(* Logix 5000 project; controller PBS_Perfusion vendor 1 type 14 code 217 rev 32.14; software revision 32.03; part 24 of 27 *)
(* tags used below, declared in another part *)
   Inp_Ready : BOOL;   // 1=Drive is ready to run
   Inp_CommandDir : BOOL;   // 1=Drive is commanded Forward, 0=Drive is commanded Reverse
   Inp_ActualDir : BOOL;   // 1=Drive is running Forward, 0=Drive is running Reverse
   Inp_FwdPermOK : BOOL;   // 1=Permissives OK, drive can start Forward
   Inp_FwdNBPermOK : BOOL;   // 1=Non-Bypassable Permissives OK, drive can start Forward
   Inp_RevPermOK : BOOL;   // 1=Permissives OK, drive can start Reverse
   Inp_RevNBPermOK : BOOL;   // 1=Non-Bypassable Permissives OK, motor can start Reverse
   Inp_IntlkOK : BOOL;   // 1=Interlocks OK, drive can start/run
   Inp_NBIntlkOK : BOOL;   // 1=Non-Bypassable Interlocks OK, drive can start/run
   Inp_OvrdCmd : DINT;   // Override Command: 0=None, 1=Stop, 2=Start Fwd 3=Start Rev
   Cfg_HasReverse : BOOL;   // 1=Drive can be run reverse, 0=Forward only
   Cfg_HasIntlkObj : BOOL;   // 1=Tells HMI a P_Intlk is connected to Inp_Intlk
   Cfg_SetTrack : BOOL;   // 1=Settings track for unselected sources, 0=no tracking
   Cfg_ShedOnFailToStart : BOOL;   // 1=Stop Motor and Alarm on Fail to Start; 0=Alarm only on Fail to Start
   Cfg_ShedOnIOFault : BOOL;   // 1=Stop Motor and Alarm on I/O Fault; 0=Alarm only on I/O Fault
   Cfg_DecPlcs : DINT;   // Number of decimal places for speed ref/fdbk display (0..6)
   Cfg_InpDLDecPlcs : DINT;   // Number of decimal places for Input Datalink display (0..6)
   Cfg_OutDLDecPlcs : DINT;   // Number of decimal places for Output Datalink display (0..6)
   Cfg_FailToStartAckReqd : ALIAS FOR FailToStart.Cfg_AckReqd;   // 1=Acknowledge required for Fail to Start Alarm
   Cfg_FailToStopAckReqd : ALIAS FOR FailToStop.Cfg_AckReqd;   // 1=Acknowledge required for Fail to Stop Alarm
   Cfg_IntlkTripAckReqd : ALIAS FOR IntlkTrip.Cfg_AckReqd;   // 1=Acknowledge required for Interlock Trip Alarm
   Cfg_DriveFaultAckReqd : ALIAS FOR DriveFault.Cfg_AckReqd;   // 1=Acknowledge required for Drive Fault Alarm
   Cfg_IOFaultAckReqd : ALIAS FOR IOFault.Cfg_AckReqd;   // 1=Acknowledge required for I/O Fault Alarm
   Cfg_FailToStartSeverity : ALIAS FOR FailToStart.Cfg_Severity;   // Fail To Start Alarm Severity: 1..250=Low, 251..500=Medium, 501..750=High, 751..1000=Urgent
   Cfg_FailToStopSeverity : ALIAS FOR FailToStop.Cfg_Severity;   // Fail To Stop Alarm Severity: 1..250=Low, 251..500=Medium, 501..750=High, 751..1000=Urgent
   Cfg_IntlkTripSeverity : ALIAS FOR IntlkTrip.Cfg_Severity;   // Interlock Trip Alarm Severity: 1..250=Low, 251..500=Medium, 501..750=High, 751..1000=Urgent
   Cfg_DriveFaultSeverity : ALIAS FOR DriveFault.Cfg_Severity;   // Drive Fault Alarm Severity: 1..250=Low, 251..500=Medium, 501..750=High, 751..1000=Urgent
   Cfg_IOFaultSeverity : ALIAS FOR IOFault.Cfg_Severity;   // I/O Fault Alarm Severity: 1..250=Low, 251..500=Medium, 501..750=High, 751..1000=Urgent
   Cfg_MaxSpdRef : REAL;   // Maximum Speed Reference in EU (for limiting)
   Cfg_SpeedRefRawMax : REAL;   // Speed Reference Maximum in Drive (raw) Units (for scaling)
   Cfg_SpeedRefEUMax : REAL;   // Speed Reference Maximum in Engineering Units (for scaling)
   Cfg_SpeedFdbkRawMax : REAL;   // Speed Feedback Maximum in Drive (raw) Units (for scaling)
   Cfg_SpeedFdbkEUMax : REAL;   // Speed Feedback Maximum in Engineering Units (for scaling)
   Cfg_InpDatalinkRawMax : REAL;   // Input Datalink Maximum in Drive (raw) Units (for scaling)
   Cfg_InpDatalinkEUMax : REAL;   // Input Datalink Maximum in Engineering Units (for scaling)
   Cfg_OutDatalinkMax : REAL;   // Maximum Output Datalink in EU (for limiting)
   Cfg_OutDatalinkRawMax : REAL;   // Output Datalink Maximum in Drive (raw) Units (for scaling)
   Cfg_OutDatalinkEUMax : REAL;   // Output Datalink Maximum in Engineering Units (for scaling)
   Cfg_SimRampT : REAL;   // Time to ramp speed fdbk when in Simulation (sec)
   Cfg_FailToStartT : REAL;   // Time after Start to get Run Feedback before Fault (sec)
   Cfg_FailToStopT : REAL;   // Time after Stop to drop Run Feedback before Fault (sec)
   Cfg_ResetPulseT : REAL;   // Time to pulse Out_Reset to clear drive fault
   Cfg_OperKeep : SINT;   // Oper keeps control in Prog / Ext: .0=Reference, .1=Start/Stop/Fwd/ Rev, .3=OutDatalink
   Cfg_ProgKeep : SINT;   // Prog keeps control in Oper / Ext: .0=Reference, .1=Start/Stop/Fwd/ Rev, .3=OutDatalink
   Cfg_ExtKeep : SINT;   // Ext keeps control in Prog / Oper: .0=Reference, .1=Start/Stop/Fwd/ Rev, .3=OutDatalink
   PSet_SpeedRef : REAL;   // Program Setting of Speed Reference (EU)
   PSet_Owner : DINT;   // Program Owner Request ID (non-zero) or Release (zero)
   XSet_SpeedRef : REAL;   // External Setting of Speed Reference (EU)
   PCmd_StartFwd : BOOL;   // Program Command to Start Drive Forward
   PCmd_StartRev : BOOL;   // Program Command to Start Drive Reverse
   PCmd_Stop : BOOL;   // Program Command to Stop Drive
   PCmd_Reset : BOOL;   // Program Command to Reset drive fault and all Alarms requiring Reset
   XCmd_StartFwd : BOOL;   // External Command to Start Drive Forward
   XCmd_StartRev : BOOL;   // External Command to Start Drive Reverse
   XCmd_Stop : BOOL;   // External Command to Stop Drive
   XCmd_JogFwd : BOOL;   // External Command to Jog Drive Forward
   XCmd_JogRev : BOOL;   // External Command to Jog Drive Reverse
   XCmd_Reset : BOOL;   // Ext Cmd to clear shed latches and cleared alarms
   Out_SpeedRef : REAL;   // Drive Speed Reference in Drive Units (typ. 0-32767 = 0 to max freq.)
   Out_Datalink : REAL;   // Auxiliary Signal (datalink) Output in Drive (raw) Units
   Out_Run : BOOL;   // 1=Start/Run Drive, 0=Stop Drive (for held starter type)
   Out_Stop : BOOL;   // 1=Stop Drive, 0=drive left in current state
   Out_Start : BOOL;   // 1=Start Drive, 0=drive left in current state
   Out_Jog : BOOL;   // 1=Jog drive at Jog Speed, -->0=stop jogging
   Out_ClearFault : BOOL;   // 1=Attempt to clear Drive Fault
   Out_Fwd : BOOL;   // 1=Set drive direction to Forward
   Out_Rev : BOOL;   // 1=Set drive direction to Reverse
   Out_Horn : BOOL;   // 1=Sound audible prior to commanded motor start
   Val_SpeedRef : REAL;   // Speed Reference (target) to drive
   Val_SpeedRefEUMax : REAL;   // Maximum of Speed Reference = MAX (Cfg_SpeedFdbkEUMin, Cfg_SpeedFdbkEUMax)
   Val_SpeedFdbkEUMax : REAL;   // Maximum of Speed Feedback = MAX (Cfg_SpeedFdbkEUMin, Cfg_SpeedFdbkEUMax)
   SrcQ_IO : DINT;   // Source and Quality of primary I/O (enumeration)
   SrcQ : DINT;   // Source and Quality of primary Val/Sts (enumeration)
   Val_Cmd : DINT;   // Device Command 0=None, 1=Stop, 2=StartFwd 3=StartRev 4=JogFwd 5=JogRev
   Val_Fdbk : DINT;   // Device Feedback 0=Stopped, 1=Running Fwd 2=Running Rev 3=Accelerating 4=Decelerating
   Val_Sts : DINT;   // Device Sts: 0=? 1=Stopped 2=RunFwd 3=RunRev 4=RunSlow 5=StartFwd 6=StartRev 7=StartSlow 8=JogFwd 9=JogRev 10=Stopping
   Val_NotifyAll : DINT;   // Highest Alarm prio and ack status this object + channel (enum)
   Val_UnackAlmC : DINT;   // Count of Unacknowledged Alarms
   Val_Owner : DINT;   // Current Object Owner ID (0=not owned)
   Sts_Stopped : BOOL;   // 1=Drive requested to stop and is confirmed stopped
   Sts_CommandDir : BOOL;   // 1=Drive commanded to Forward, 0=Reverse
   Sts_ActualDir : BOOL;   // 1=Drive Actual direction is Forward, 0=Reverse
   Sts_Available : BOOL;   // 1=Drive available for control by automation (Prog)
   Sts_NotRdy : BOOL;   // 1=Device Not Ready, see detail bits for reason
   Nrdy_Fail : BOOL;   // 1=Device Not Ready: Device Failure (Shed Requires Reset)
   Nrdy_Intlk : BOOL;   // 1=Device Not Ready: Interlock Not OK
   Nrdy_IOFault : BOOL;   // 1=Device Not Ready: I/O Fault (Shed Requires Reset)
   Nrdy_PrioStop : BOOL;   // 1=Device Not Ready: Oper/Ext Priority Stop Requires Reset
   Sts_MaintByp : BOOL;   // 1=A Maintenance Bypass is Active, display icon
   Sts_Prog : ALIAS FOR CmdSrc.Sts_Prog;
   Sts_Oper : ALIAS FOR CmdSrc.Sts_Oper;
   Sts_Normal : ALIAS FOR CmdSrc.Sts_Normal;
   Sts_ExtReqInh : ALIAS FOR CmdSrc.Sts_ExtReqInh;
   Sts_RdyAck : BOOL;   // 1=An alarm is ready to be acknowledged
   Ack_FailToStart : ALIAS FOR FailToStart.Ack;   // 1=Fail to Start Alarm has been acknowledged
   Ack_FailToStop : ALIAS FOR FailToStop.Ack;   // 1=Fail to Stop Alarm has been acknowledged
   Ack_IntlkTrip : ALIAS FOR IntlkTrip.Ack;   // 1=Interlock Trip Alarm has been acknowledged
   Ack_DriveFault : ALIAS FOR DriveFault.Ack;   // 1=Drive Fault Alarm has been acknowledged
   Ack_IOFault : ALIAS FOR IOFault.Ack;   // 1=I/O Fault Alarm has been acknowledged
   P_VSD : BOOL;   // Unique Parameter Name for auto - discovery
   Wrk_Run : BOOL;   // 1=Drive should be "running", 0=should be "stopped"
   Wrk_Jog : BOOL;   // 1=Jog Drive, 0=Drive not jogging
   OCmd_ResetAckAll : BOOL;   // Oper Cmd to reset shed latches and cleared alarms, plus Acknowledge alarms
   OCmd_Reset : BOOL;   // Oper Cmd to clear shed latches and cleared alarms
   OCmd_JogRev : BOOL;   // Operator Command to Jog Drive Reverse (not cleared by instruction!)
   OCmd_JogFwd : BOOL;   // Operator Command to Jog Drive Forward (not cleared by instruction!)
   OCmd_Stop : BOOL;   // Operator Command to Stop Drive
   OCmd_StartRev : BOOL;   // Operator Command to Start Drive Reverse
   OCmd_StartFwd : BOOL;   // Operator Command to Start Drive Forward
   MCmd_Check : BOOL;   // Maintenance Command to Check (not bypass) all Interlocks and Permissives
   MCmd_Bypass : BOOL;   // Maintenance Command to Bypass all Bypassable Interlocks and Permissives
   ORdy_ResetAckAll : BOOL;   // 1=Ready for OCmd_ResetAckAll (enables HMI button)
   ORdy_Reset : BOOL;   // 1=Ready for OCmd_Reset (enables HMI button)
   ORdy_JogRev : BOOL;   // 1=Ready for OCmd_JogRev (enabled HMI button)
   ORdy_JogFwd : BOOL;   // 1=Ready for OCmd_JogFwd (enables HMI button)
   ORdy_Stop : BOOL;   // 1=Ready for OCmd_Stop (enables HMI button)
   ORdy_StartRev : BOOL;   // 1=Ready for OCmd_StartRev (enables HMI button)
   ORdy_StartFwd : BOOL;   // 1=Ready for OCmd_StartFwd (enables HMI button)
   ORdy_SpeedRef : BOOL;   // 1=Ready for OSet_SpeedRef (enables data entry field)
   MRdy_Check : BOOL;   // 1=Ready for MCmd_Check (enables HMI button)
   MRdy_Bypass : BOOL;   // 1=Ready for MCmd_Bypass (enables HMI button)
(* P_VSD, continued *)

ROUTINE Prescan   (* ladder *)
// Clear Ownership, set drive to STOP, clear "lurking" Commands
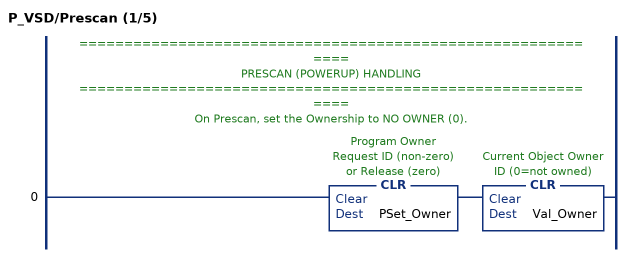
   // ============================================================
   // PRESCAN (POWERUP) HANDLING
   // ============================================================
   // On Prescan, set the Ownership to NO OWNER (0).
   0: CLR(PSet_Owner)CLR(Val_Owner);
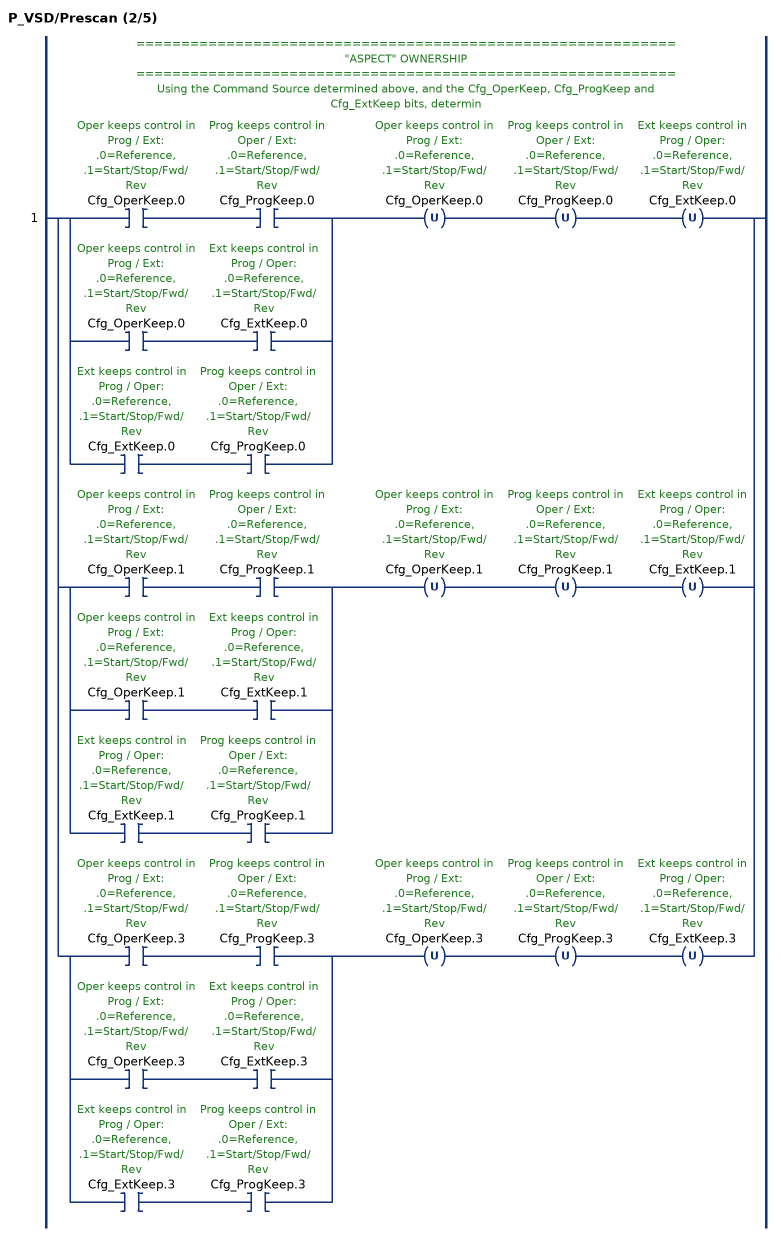
   // ============================================================
   // "ASPECT" OWNERSHIP
   // ============================================================
   // Using the Command Source determined above, and the Cfg_OperKeep, Cfg_ProgKeep and
   // Cfg_ExtKeep bits, determin
   1: [[XIC(Cfg_OperKeep.0) XIC(Cfg_ProgKeep.0) ,XIC(Cfg_OperKeep.0) XIC(Cfg_ExtKeep.0) ,XIC(Cfg_ExtKeep.0) XIC(Cfg_ProgKeep.0) ] OTU(Cfg_OperKeep.0) OTU(Cfg_ProgKeep.0) OTU(Cfg_ExtKeep.0) ,[XIC(Cfg_OperKeep.1) XIC(Cfg_ProgKeep.1) ,XIC(Cfg_OperKeep.1) XIC(Cfg_ExtKeep.1) ,XIC(Cfg_ExtKeep.1) XIC(Cfg_ProgKeep.1) ] OTU(Cfg_OperKeep.1) OTU(Cfg_ProgKeep.1) OTU(Cfg_ExtKeep.1) ,[XIC(Cfg_OperKeep.3) XIC(Cfg_ProgKeep.3) ,XIC(Cfg_OperKeep.3) XIC(Cfg_ExtKeep.3) ,XIC(Cfg_ExtKeep.3) XIC(Cfg_ProgKeep.3) ] OTU(Cfg_OperKeep.3) OTU(Cfg_ProgKeep.3) OTU(Cfg_ExtKeep.3) ];
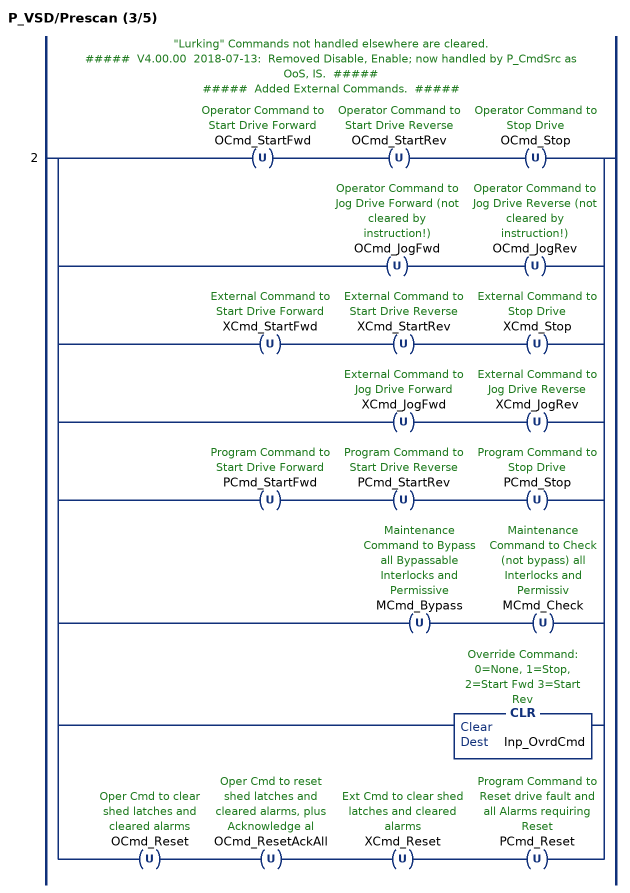
   // "Lurking" Commands not handled elsewhere are cleared.
   // #####  V4.00.00  2018-07-13:  Removed Disable, Enable; now handled by P_CmdSrc as OoS, IS.  #####
   // #####  Added External Commands.  #####
   2: [OTU(OCmd_StartFwd) OTU(OCmd_StartRev) OTU(OCmd_Stop) ,OTU(OCmd_JogFwd) OTU(OCmd_JogRev) ,OTU(XCmd_StartFwd) OTU(XCmd_StartRev) OTU(XCmd_Stop) ,OTU(XCmd_JogFwd) OTU(XCmd_JogRev) ,OTU(PCmd_StartFwd) OTU(PCmd_StartRev) OTU(PCmd_Stop) ,OTU(MCmd_Bypass) OTU(MCmd_Check) ,CLR(Inp_OvrdCmd) ,OTU(OCmd_Reset) OTU(OCmd_ResetAckAll) OTU(XCmd_Reset) OTU(PCmd_Reset) ];
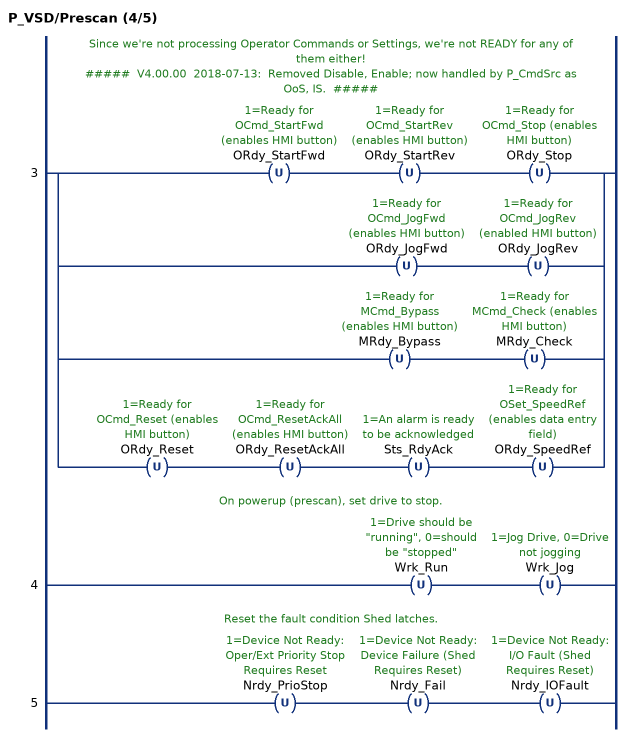
   // Since we're not processing Operator Commands or Settings, we're not READY for any of them either!
   // #####  V4.00.00  2018-07-13:  Removed Disable, Enable; now handled by P_CmdSrc as OoS, IS.  #####
   3: [OTU(ORdy_StartFwd) OTU(ORdy_StartRev) OTU(ORdy_Stop) ,OTU(ORdy_JogFwd) OTU(ORdy_JogRev) ,OTU(MRdy_Bypass) OTU(MRdy_Check) ,OTU(ORdy_Reset) OTU(ORdy_ResetAckAll) OTU(Sts_RdyAck) OTU(ORdy_SpeedRef) ];
   // On powerup (prescan), set drive to stop.
   4: OTU(Wrk_Run)OTU(Wrk_Jog);
   // Reset the fault condition Shed latches.
   5: OTU(Nrdy_PrioStop)OTU(Nrdy_Fail)OTU(Nrdy_IOFault);
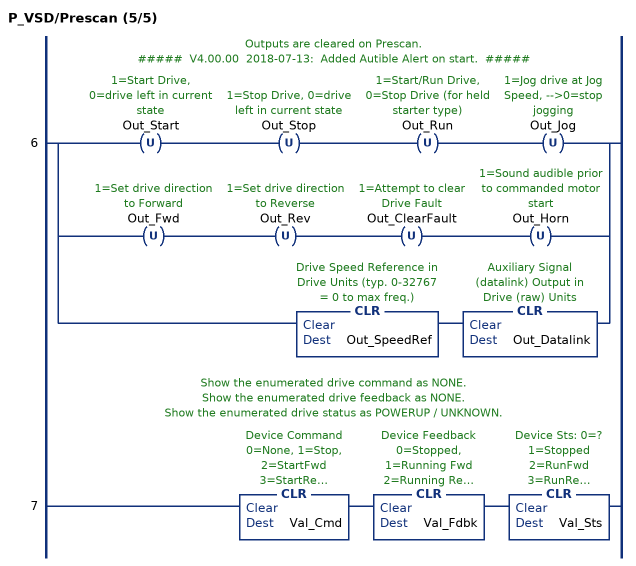
   // Outputs are cleared on Prescan.
   // #####  V4.00.00  2018-07-13:  Added Autible Alert on start.  #####
   6: [OTU(Out_Start) OTU(Out_Stop) OTU(Out_Run) OTU(Out_Jog) ,OTU(Out_Fwd) OTU(Out_Rev) OTU(Out_ClearFault) OTU(Out_Horn) ,CLR(Out_SpeedRef) CLR(Out_Datalink) ];
   // Show the enumerated drive command as NONE.
   // Show the enumerated drive feedback as NONE.
   // Show the enumerated drive status as POWERUP / UNKNOWN.
   7: CLR(Val_Cmd)CLR(Val_Fdbk)CLR(Val_Sts);
END_ROUTINE
END_ADD_ON_INSTRUCTION

ADD_ON_INSTRUCTION PBS_error   (* revision 1.0 *)
VAR_INPUT
   errorInteger : INT; {required}
END_VAR
VAR_OUTPUT
   OK : BOOL; {access Read Only, visible}
   Failure : BOOL; {access Read Only, visible}
   HiHi : BOOL; {access Read Only, visible}
   Hi : BOOL; {access Read Only, visible}
   Lo : BOOL; {access Read Only, visible}
   LoLo : BOOL; {access Read Only, visible}
END_VAR

ROUTINE Logic   (* ladder *)
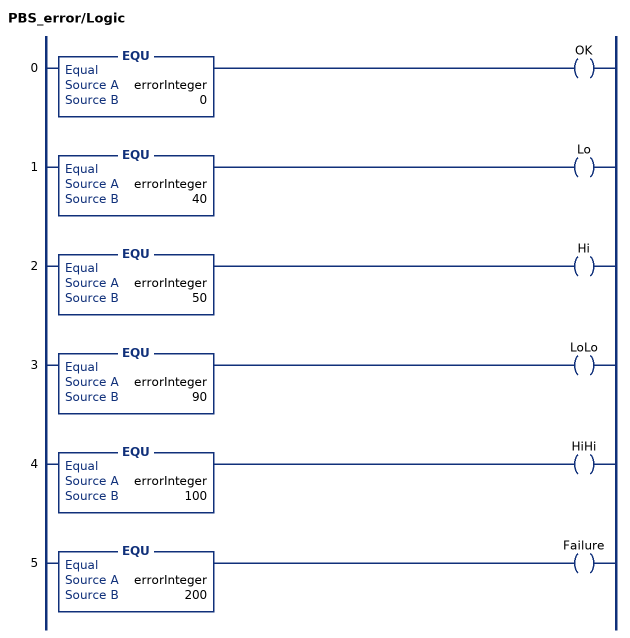
   0: EQU(errorInteger,0)OTE(OK);
   1: EQU(errorInteger,40)OTE(Lo);
   2: EQU(errorInteger,50)OTE(Hi);
   3: EQU(errorInteger,90)OTE(LoLo);
   4: EQU(errorInteger,100)OTE(HiHi);
   5: EQU(errorInteger,200)OTE(Failure);
END_ROUTINE
END_ADD_ON_INSTRUCTION

ADD_ON_INSTRUCTION Pump_Cal   (* revision 1.3, vendor JES Inc. *)
// Pump Calibration Module
// Revision note:
// 1.0 Published
// 1.1 Using the P_VSD block
// 1.2 Included Pump Cal into the AOI
// 1,3 Modified to include native PlantPax VSD Block
VAR_INPUT
   Cal_CollectionType : BOOL;   // 0 = Mass, 1 = Volume
   Cal_CollectedQuantity : REAL;   // Operator Input Collected Mass or Volume obtained
   Cal_Density : REAL;   // Operator Input Density (g/ml)
   Cal_Duration : REAL;   // Operator Input pump run duration (min)
   Cal_PumpSpeed : REAL;   // Set Pump Speed in %
   Cal_CmdStart : BOOL;   // Start Cal Sequence
   Cal_CmdStop : BOOL;   // Stop/Abort Cal Sequence
END_VAR
VAR_OUTPUT
   Cal_Aborted : BOOL; {access Read Only}   // Calibration Sequence is Aborted
   Cal_Complete : BOOL; {access Read Only}   // Calibration Sequence is Complete
   Cal_Running : BOOL; {access Read Only}   // Calibration Sequence is Active
   Cal_EUMax : REAL; {access Read Only}   // Calculated max EU (mL/min)
   Cal_Phase2Active : BOOL; {access Read Only}   // Cal Pump run complete, now calculating Pump EU Max
END_VAR
VAR_INPUT
   Cal_CmdPhase2Accept : BOOL;   // Accept button pressed by Operator after inputing collected volume or mass
END_VAR
VAR_OUTPUT
   Cal_Started : BOOL; {access Read Only}
   Cal_Runtime : REAL; {access Read Only}   // Accumulation time converted to minutes -For HMI-
END_VAR
VAR_IN_OUT
   Drive_Sts_RunningFwd : BOOL; {required}
   Drive_PCmd_Prog : BOOL; {required}
   Drive_Cfg_SpeedRefEUMin : REAL; {required}
   Drive_Cfg_SpeedRefEUMax : REAL; {required}
   Drive_Cfg_SpeedFdbkEUMin : REAL; {required}
   Drive_Cfg_SpeedFdbkEUMax : REAL; {required}
   Drive_Cfg_MinSpdRef : REAL; {required}
   Drive_Cfg_MaxSpdRef : REAL; {required}
   Drive_PSet_SpeedRef : REAL; {required}
   Drive_PCmd_StartFwd : BOOL; {required}
   Drive_Sts_Prog : BOOL; {required}
   Drive_PCmd_Stop : BOOL; {required}
END_VAR
VAR
   ONS : DINT; {access None}
   Cal_RunTimer2 : TIMER; {access None}   // Run Timer used to calculate how long the pump is running
   Cal_RunTimer : TIMER; {access None}
   Cal_CalculatedVol : REAL; {access Read Only}   // Internal calculated volume if the operator selected volume
END_VAR

ROUTINE Logic   (* ladder *)
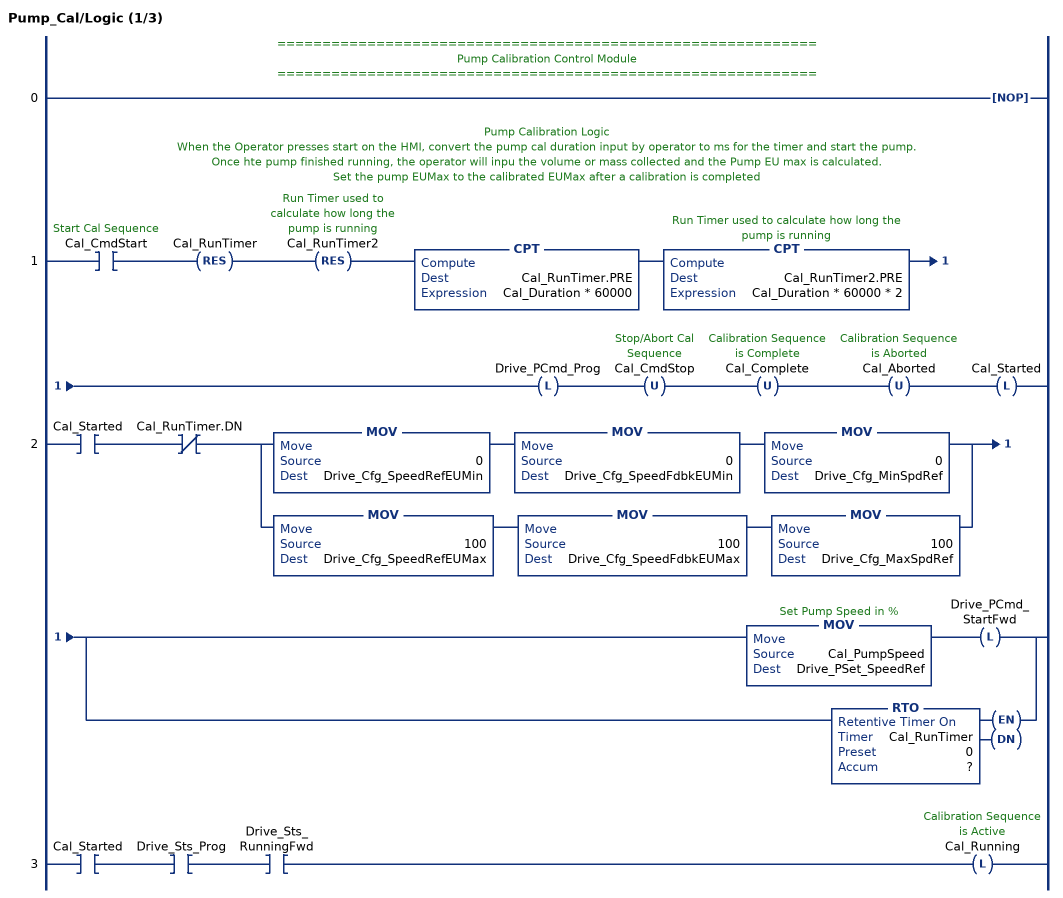
   // ============================================================
   // Pump Calibration Control Module
   // ============================================================
   0: NOP();
   // Pump Calibration Logic
   // When the Operator presses start on the HMI, convert the pump cal duration input by operator to ms for the timer and start the pump.
   // Once hte pump finished running, the operator will inpu the volume or mass collected and the Pump EU max is calculated.
   // Set the pump EUMax to the calibrated EUMax after a calibration is completed
   1: XIC(Cal_CmdStart)RES(Cal_RunTimer)RES(Cal_RunTimer2)CPT(Cal_RunTimer.PRE,Cal_Duration * 60000)CPT(Cal_RunTimer2.PRE,Cal_Duration * 60000 * 2)OTL(Drive_PCmd_Prog)OTU(Cal_CmdStop)OTU(Cal_Complete)OTU(Cal_Aborted)OTL(Cal_Started);
   2: XIC(Cal_Started)XIO(Cal_RunTimer.DN)[MOV(0,Drive_Cfg_SpeedRefEUMin) MOV(0,Drive_Cfg_SpeedFdbkEUMin) MOV(0,Drive_Cfg_MinSpdRef) ,MOV(100,Drive_Cfg_SpeedRefEUMax) MOV(100,Drive_Cfg_SpeedFdbkEUMax) MOV(100,Drive_Cfg_MaxSpdRef) ][MOV(Cal_PumpSpeed,Drive_PSet_SpeedRef) OTL(Drive_PCmd_StartFwd) ,RTO(Cal_RunTimer,?,?) ];
   3: XIC(Cal_Started)XIC(Drive_Sts_Prog)XIC(Drive_Sts_RunningFwd)OTL(Cal_Running);
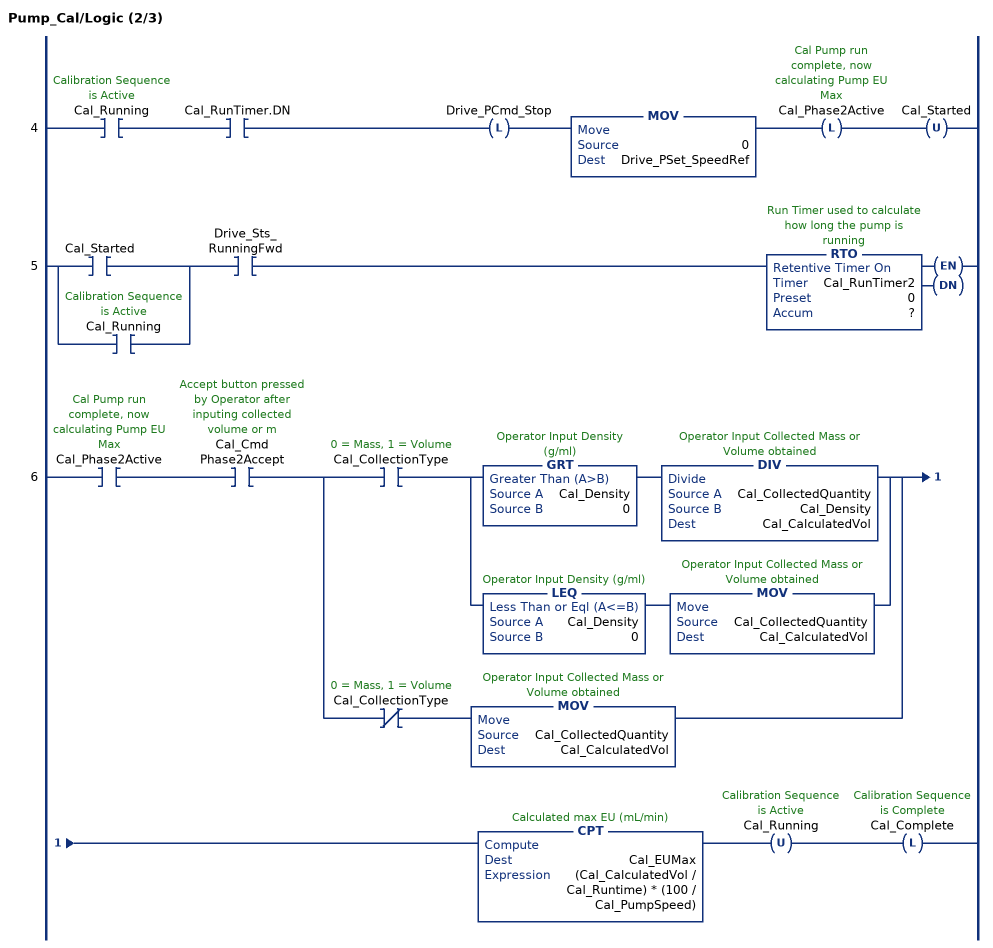
   4: XIC(Cal_Running)XIC(Cal_RunTimer.DN)OTL(Drive_PCmd_Stop)MOV(0,Drive_PSet_SpeedRef)OTL(Cal_Phase2Active)OTU(Cal_Started);
   5: [XIC(Cal_Started) ,XIC(Cal_Running) ]XIC(Drive_Sts_RunningFwd)RTO(Cal_RunTimer2,?,?);
   6: XIC(Cal_Phase2Active)XIC(Cal_CmdPhase2Accept)[XIC(Cal_CollectionType) [GRT(Cal_Density,0) DIV(Cal_CollectedQuantity,Cal_Density,Cal_CalculatedVol) ,LEQ(Cal_Density,0) MOV(Cal_CollectedQuantity,Cal_CalculatedVol) ] ,XIO(Cal_CollectionType) MOV(Cal_CollectedQuantity,Cal_CalculatedVol) ]CPT(Cal_EUMax,(Cal_CalculatedVol / Cal_Runtime) * (100 / Cal_PumpSpeed))OTU(Cal_Running)OTL(Cal_Complete);
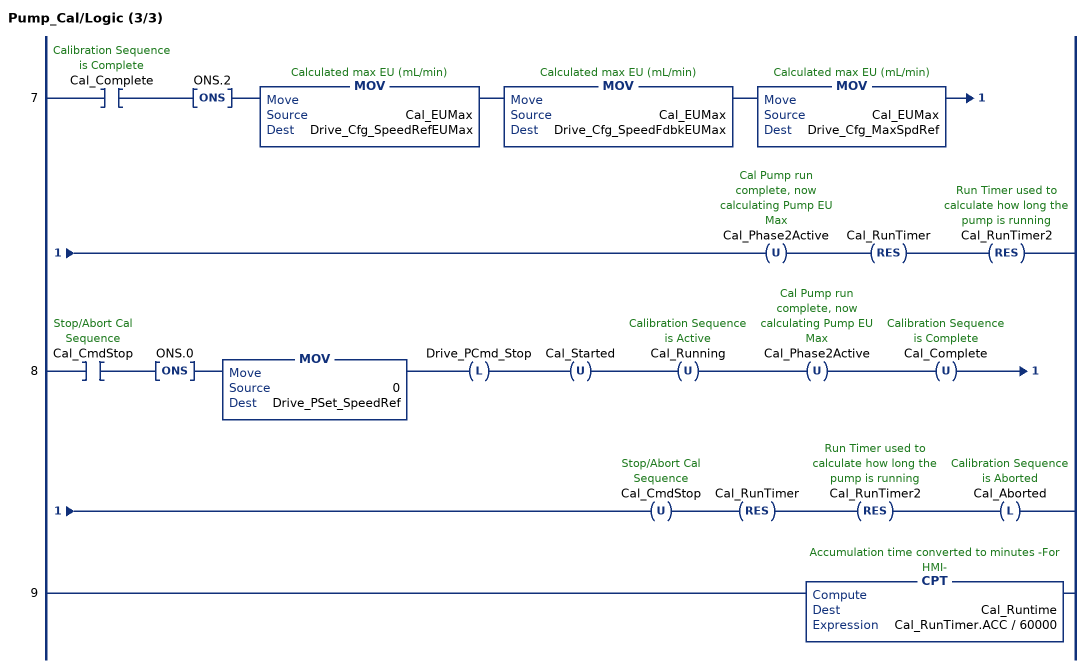
   7: XIC(Cal_Complete)ONS(ONS.2)MOV(Cal_EUMax,Drive_Cfg_SpeedRefEUMax)MOV(Cal_EUMax,Drive_Cfg_SpeedFdbkEUMax)MOV(Cal_EUMax,Drive_Cfg_MaxSpdRef)OTU(Cal_Phase2Active)RES(Cal_RunTimer)RES(Cal_RunTimer2);
   8: XIC(Cal_CmdStop)ONS(ONS.0)MOV(0,Drive_PSet_SpeedRef)OTL(Drive_PCmd_Stop)OTU(Cal_Started)OTU(Cal_Running)OTU(Cal_Phase2Active)OTU(Cal_Complete)OTU(Cal_CmdStop)RES(Cal_RunTimer)RES(Cal_RunTimer2)OTL(Cal_Aborted);
   9: CPT(Cal_Runtime,Cal_RunTimer.ACC / 60000);
END_ROUTINE
END_ADD_ON_INSTRUCTION

VAR_GLOBAL   (* controller tags *)
   AIC0706 : PID_ENHANCED := (PV := 3.2633398, PVEUMax := 200.0, SPProg := 90.0, SPOper := 3.2633398, SPHLimit := 200.0, RatioProg := 1.0, RatioOper := 1.0, RatioHLimit := 1.0, RatioLLimit := 1.0, CVEUMax := 100.0, CVHLimit := 100.0, CVROCLimit := 2.0, PGain := 1.0, IGain := 0.5, PVEDerivative := 1, PVTracking := 1, DevHHLimit := 50.0, DevHLimit := 25.0, DevLLimit := 25.0, DevLLLimit := 50.0, RTSTime := 1, SP := 3.2633398, SPPercent := 1.6316699, PVPercent := 1.6316699, InitPrimary := 1, Ratio := 1.0, ProgOper := 1, Manual := 1, DeltaT := 1.0);   // Disolved Oxygen PID
   AIC0707 : PID_ENHANCED := (PV := -9998.96, PVEUMax := 8.5, PVEUMin := 5.5, SPProg := 8.0, SPOper := 5.5, SPHLimit := 8.5, SPLLimit := 5.5, RatioProg := 1.0, RatioOper := 1.0, RatioHLimit := 1.0, RatioLLimit := 1.0, CVInitValue := 50.0, CVProg := 50.0, CVOper := 50.0, CVOverride := 50.0, CVEUMax := 100.0, CVHLimit := 100.0, CVROCLimit := 2.0, PGain := 2.0, IGain := 1.0, PVEDerivative := 1, PVTracking := 1, DevHHLimit := 0.5, DevHLimit := 0.3, DevLLimit := 0.3, DevLLLimit := 0.5, RTSTime := 1, CVEU := 50.0, CV := 50.0, SP := 5.5, SPLAlarm := 1, PVPercent := -333482.0, E := 10004.46, EPercent := 333482.0, InitPrimary := 1, WindupLOut := 1, Ratio := 1.0, DevLAlarm := 1, DevLLAlarm := 1, ProgOper := 1, Manual := 1, DeltaT := 1.0);   // ph PID
   AIC703 : P_AInAdv := (Inp_HiHiGate := 1, Inp_HiGate := 1, Inp_LoGate := 1, Inp_LoLoGate := 1, Inp_HiRoCGate := 1, Inp_HiDevGate := 1, Inp_LoDevGate := 1, Inp_FailGate := 1, Cfg_PVDecPlcs := 2, Cfg_HiHiAckReqd := 1, Cfg_HiAckReqd := 1, Cfg_LoAckReqd := 1, Cfg_LoLoAckReqd := 1, Cfg_HiRoCAckReqd := 1, Cfg_HiDevAckReqd := 1, Cfg_LoDevAckReqd := 1, Cfg_FailAckReqd := 1, Cfg_HiHiSeverity := 750, Cfg_HiSeverity := 500, Cfg_LoSeverity := 500, Cfg_LoLoSeverity := 750, Cfg_HiRoCSeverity := 500, Cfg_HiDevSeverity := 500, Cfg_LoDevSeverity := 500, Cfg_FailSeverity := 1000, Cfg_InpRawMax := 100.0, Cfg_PVEUMax := 100.0, Cfg_RateTime := 1.0, Cfg_CtrlHiHiLim := 1.5e+38, Cfg_CtrlHiHiDB := 1.0, Cfg_CtrlHiLim := 1.5e+38, Cfg_CtrlHiDB := 1.0, Cfg_CtrlLoLim := -1.5e+38, Cfg_CtrlLoDB := 1.0, Cfg_CtrlLoLoLim := -1.5e+38, Cfg_CtrlLoLoDB := 1.0, Cfg_HiHiLim := 1.5e+38, Cfg_HiHiDB := 1.0, Cfg_HiLim := 1.5e+38, Cfg_HiDB := 1.0, Cfg_LoLim := -1.5e+38, Cfg_LoDB := 1.0, Cfg_LoLoLim := -1.5e+38, Cfg_LoLoDB := 1.0, Cfg_HiRoCLim := 1.5e+38, Cfg_HiRoCDB := 1.0, Cfg_HiDevLim := 1.5e+38, Cfg_HiDevDB := 1.0, Cfg_LoDevLim := -1.5e+38, Cfg_LoDevDB := 1.0, Cfg_FailHiLim := 103.958336, Cfg_FailLoLim := -2.0833333, Cfg_FailDB := 0.41666666, MSet_SubstPV := 10.0, Val := 10.0, Val_PVMinCapt := 10.0, Val_PVMaxCapt := 10.0, Val_PVEUMax := 100.0, SrcQ_IO := 1, SrcQ := 18,
        Sts_SubstPV := 1, Sts_MaintByp := 1, Sts_HiHiGate := 1, Ack_HiHi := 1, Sts_HiGate := 1, Ack_Hi := 1, Sts_LoGate := 1, Ack_Lo := 1, Sts_LoLoGate := 1, Ack_LoLo := 1, Sts_HiRoCGate := 1, Ack_HiRoC := 1, Sts_HiDevGate := 1, Ack_HiDev := 1, Sts_LoDevGate := 1, Ack_LoDev := 1, Sts_FailGate := 1, Ack_Fail := 1);   // BRX DO PV
   AirManualSP : REAL;
   AirPercentOut : REAL := 0.95;
   AirProgOper : BOOL := 1;
   AT701 : P_AInAdv := (Inp_HiHiGate := 1, Inp_HiGate := 1, Inp_LoGate := 1, Inp_LoLoGate := 1, Inp_HiRoCGate := 1, Inp_HiDevGate := 1, Inp_LoDevGate := 1, Inp_FailGate := 1, Cfg_PVDecPlcs := 2, Cfg_HiHiAckReqd := 1, Cfg_HiAckReqd := 1, Cfg_LoAckReqd := 1, Cfg_LoLoAckReqd := 1, Cfg_HiRoCAckReqd := 1, Cfg_HiDevAckReqd := 1, Cfg_LoDevAckReqd := 1, Cfg_FailAckReqd := 1, Cfg_HiHiSeverity := 750, Cfg_HiSeverity := 500, Cfg_LoSeverity := 500, Cfg_LoLoSeverity := 750, Cfg_HiRoCSeverity := 500, Cfg_HiDevSeverity := 500, Cfg_LoDevSeverity := 500, Cfg_FailSeverity := 1000, Cfg_InpRawMax := 100.0, Cfg_PVEUMax := 100.0, Cfg_RateTime := 1.0, Cfg_CtrlHiHiLim := 1.5e+38, Cfg_CtrlHiHiDB := 1.0, Cfg_CtrlHiLim := 1.5e+38, Cfg_CtrlHiDB := 1.0, Cfg_CtrlLoLim := -1.5e+38, Cfg_CtrlLoDB := 1.0, Cfg_CtrlLoLoLim := -1.5e+38, Cfg_CtrlLoLoDB := 1.0, Cfg_HiHiLim := 1.5e+38, Cfg_HiHiDB := 1.0, Cfg_HiLim := 1.5e+38, Cfg_HiDB := 1.0, Cfg_LoLim := -1.5e+38, Cfg_LoDB := 1.0, Cfg_LoLoLim := -1.5e+38, Cfg_LoLoDB := 1.0, Cfg_HiRoCLim := 1.5e+38, Cfg_HiRoCDB := 1.0, Cfg_HiDevLim := 1.5e+38, Cfg_HiDevDB := 1.0, Cfg_LoDevLim := -1.5e+38, Cfg_LoDevDB := 1.0, Cfg_FailHiLim := 103.958336, Cfg_FailLoLim := -2.0833333, Cfg_FailDB := 0.41666666, MSet_SubstPV := 12.0, Val := 12.0, Val_PVMinCapt := 12.0, Val_PVMaxCapt := 12.0, Val_PVEUMax := 100.0, SrcQ_IO := 1, SrcQ := 18,
        Sts_SubstPV := 1, Sts_MaintByp := 1, Sts_HiHiGate := 1, Ack_HiHi := 1, Sts_HiGate := 1, Ack_Hi := 1, Sts_LoGate := 1, Ack_Lo := 1, Sts_LoLoGate := 1, Ack_LoLo := 1, Sts_HiRoCGate := 1, Ack_HiRoC := 1, Sts_HiDevGate := 1, Ack_HiDev := 1, Sts_LoDevGate := 1, Ack_LoDev := 1, Sts_FailGate := 1, Ack_Fail := 1);   // DO Transmitter
   AT702 : P_AInAdv := (Inp_HiHiGate := 1, Inp_HiGate := 1, Inp_LoGate := 1, Inp_LoLoGate := 1, Inp_HiRoCGate := 1, Inp_HiDevGate := 1, Inp_LoDevGate := 1, Inp_FailGate := 1, Cfg_PVDecPlcs := 3, Cfg_HiHiAckReqd := 1, Cfg_HiAckReqd := 1, Cfg_LoAckReqd := 1, Cfg_LoLoAckReqd := 1, Cfg_HiRoCAckReqd := 1, Cfg_HiDevAckReqd := 1, Cfg_LoDevAckReqd := 1, Cfg_FailAckReqd := 1, Cfg_HiHiSeverity := 750, Cfg_HiSeverity := 500, Cfg_LoSeverity := 500, Cfg_LoLoSeverity := 750, Cfg_HiRoCSeverity := 500, Cfg_HiDevSeverity := 500, Cfg_LoDevSeverity := 500, Cfg_FailSeverity := 1000, Cfg_InpRawMax := 100.0, Cfg_PVEUMax := 14.0, Cfg_RateTime := 1.0, Cfg_CtrlHiHiLim := 1.5e+38, Cfg_CtrlHiHiDB := 1.0, Cfg_CtrlHiLim := 1.5e+38, Cfg_CtrlHiDB := 1.0, Cfg_CtrlLoLim := -1.5e+38, Cfg_CtrlLoDB := 1.0, Cfg_CtrlLoLoLim := -1.5e+38, Cfg_CtrlLoLoDB := 1.0, Cfg_HiHiLim := 1.5e+38, Cfg_HiHiDB := 1.0, Cfg_HiLim := 1.5e+38, Cfg_HiDB := 1.0, Cfg_LoLim := -1.5e+38, Cfg_LoDB := 1.0, Cfg_LoLoLim := -1.5e+38, Cfg_LoLoDB := 1.0, Cfg_HiRoCLim := 1.5e+38, Cfg_HiRoCDB := 1.0, Cfg_HiDevLim := 1.5e+38, Cfg_HiDevDB := 1.0, Cfg_LoDevLim := -1.5e+38, Cfg_LoDevDB := 1.0, Cfg_FailHiLim := 103.958336, Cfg_FailLoLim := -2.0833333, Cfg_FailDB := 0.41666666, MSet_SubstPV := 7.2, Val := 7.2, Val_PVMinCapt := 7.2, Val_PVMaxCapt := 7.2, Val_PVEUMax := 14.0, SrcQ_IO := 1, SrcQ := 18,
        Sts_SubstPV := 1, Sts_MaintByp := 1, Sts_HiHiGate := 1, Ack_HiHi := 1, Sts_HiGate := 1, Ack_Hi := 1, Sts_LoGate := 1, Ack_Lo := 1, Sts_LoLoGate := 1, Ack_LoLo := 1, Sts_HiRoCGate := 1, Ack_HiRoC := 1, Sts_HiDevGate := 1, Ack_HiDev := 1, Sts_LoDevGate := 1, Ack_LoDev := 1, Sts_FailGate := 1, Ack_Fail := 1);   // pH Transmitter
   BOR_1 : FBD_BOOLEAN_OR;
   BOR_2 : FBD_BOOLEAN_OR;
   BOR_3 : FBD_BOOLEAN_OR;
   BOR_4 : FBD_BOOLEAN_OR;
   BOR_5 : FBD_BOOLEAN_OR;
   BRX_Comm_Toggle : BOOL;
   BRX_Data : PBSdata_UDT := (jsonFailure := 1);
   Brx_heartbeat_Alarm : BOOL;
   Brx_Heartbeat_Alarm_Reset : BOOL;
   BRX_Heartbeat_Fail : TIMER := (PRE := 10000);
   BRX_HiAdj : BOOL;   // BRX HI adj in progress
   BRX_HiAdjEnable : BOOL := 1;
   BRX_HiAdjTimer : TIMER := (PRE := 15000);
   BRX_HiadjTimeSP : REAL := 15.0;
   BRX_HiSP : REAL := 60.0;
   BRX_Level_EUMax : REAL := 1.1;
   BRX_Level_EUmin : REAL := 0.9;
   BRX_Level_Initialize : BOOL := 1;
   BRX_Level_RawMax : REAL := 100.0;
   BRX_Level_RawMin : REAL;
   BRX_Level_Scaler : SCALE := (In := 50.0, InRawMax := 100.0, InEUMax := 1.1, InEUMin := 0.9, Out := 1.0);
   BRX_LevelPID : PID_ENHANCED := (PV := 4.3, PVEUMax := 100.0, SPOper := 5.0, SPHLimit := 100.0, RatioProg := 1.0, RatioOper := 1.0, RatioHLimit := 1.0, RatioLLimit := 1.0, CVInitReq := 1, CVInitValue := 50.0, CVOper := 50.0, CVPrevious := 50.0, CVEUMax := 100.0, CVHLimit := 100.0, ControlAction := 1, PGain := 2.0, IGain := 5.0, PVEDerivative := 1, ProgOperReq := 1, ProgAutoReq := 1, RTSTime := 1, CVEU := 50.0, CV := 50.0, CVInitializing := 1, SP := 5.0, SPPercent := 5.0, PVPercent := 4.3, E := -0.6999998, EPercent := -0.6999998, InitPrimary := 1, Ratio := 1.0, Auto := 1, DeltaT := 1.0);
   BRX_LoAdj : BOOL;   // BRX Lo Adj in progress
   BRX_LoAdjEnable : BOOL := 1;
   BRX_LoAdjTimer : TIMER := (PRE := 5000);
   BRX_LoadjTimeSP : REAL := 5.0;
   BRX_LoSP : REAL := 9.0;
   C02Scaler : SCALE := (InRawMax := 100.0, InEUMax := 0.083330005, Limiting := 1);
   C02Scaler1 : SCALE;
   CCA_3way : P_D4SD := (Inp_PermOK0 := 1, Inp_NBPermOK0 := 1, Inp_PermOK1 := 1, Inp_NBPermOK1 := 1, Inp_PermOK2 := 1, Inp_NBPermOK2 := 1, Inp_PermOK3 := 1, Inp_NBPermOK3 := 1, Inp_IntlkOK := 1, Inp_NBIntlkOK := 1, Cfg_NumStates := 2, Cfg_OutSt0Write := 2#0000_1111, Cfg_OutSt0State := 2#0000_0001, Cfg_OutSt1Write := 2#0000_1111, Cfg_OutSt1State := 2#0000_0010, Cfg_OutSt2Write := 2#0000_1111, Cfg_OutSt2State := 2#0000_0100, Cfg_OutSt3Write := 2#0000_1111, Cfg_OutSt3State := 2#0000_1000, Cfg_FdbkSt0State := 2#0000_0001, Cfg_FdbkSt1State := 2#0000_0010, Cfg_FdbkSt2State := 2#0000_0100, Cfg_FdbkSt3State := 2#0000_1000, Cfg_FailAckReqd := 1, Cfg_DeviceFaultAckReqd := 1, Cfg_IntlkTripAckReqd := 1, Cfg_IOFaultAckReqd := 1, Cfg_FailSeverity := 1000, Cfg_DeviceFaultSeverity := 1000, Cfg_IntlkTripSeverity := 500, Cfg_IOFaultSeverity := 1000, Cfg_SimFdbkT := 2.0, Cfg_FailT := 10.0, SrcQ_IO := 2, SrcQ := 2, Val_Sts := 1, Sts_St0 := 1, Sts_Oper := 1, Sts_Normal := 1, Sts_ExtReqInh := 1, Ack_Fail := 1, Ack_DeviceFault := 1, Ack_IntlkTrip := 1, Ack_IOFault := 1);   // TIE IO TO STATUS BITS NOT OUTPUT BITS ON p_d4sd for all 4 of them, otherwise will not hold position through power cycle
   CCAMaxCalc : REAL := 0.33333334;
   CO2_3way : P_D4SD := (Inp_PermOK0 := 1, Inp_NBPermOK0 := 1, Inp_PermOK1 := 1, Inp_NBPermOK1 := 1, Inp_PermOK2 := 1, Inp_NBPermOK2 := 1, Inp_PermOK3 := 1, Inp_NBPermOK3 := 1, Inp_IntlkOK := 1, Inp_NBIntlkOK := 1, Cfg_NumStates := 2, Cfg_OutSt0Write := 2#0000_1111, Cfg_OutSt0State := 2#0000_0001, Cfg_OutSt1Write := 2#0000_1111, Cfg_OutSt1State := 2#0000_0010, Cfg_OutSt2Write := 2#0000_1111, Cfg_OutSt2State := 2#0000_0100, Cfg_OutSt3Write := 2#0000_1111, Cfg_OutSt3State := 2#0000_1000, Cfg_FdbkSt0State := 2#0000_0001, Cfg_FdbkSt1State := 2#0000_0010, Cfg_FdbkSt2State := 2#0000_0100, Cfg_FdbkSt3State := 2#0000_1000, Cfg_FailAckReqd := 1, Cfg_DeviceFaultAckReqd := 1, Cfg_IntlkTripAckReqd := 1, Cfg_IOFaultAckReqd := 1, Cfg_FailSeverity := 1000, Cfg_DeviceFaultSeverity := 1000, Cfg_IntlkTripSeverity := 500, Cfg_IOFaultSeverity := 1000, Cfg_SimFdbkT := 2.0, Cfg_FailT := 10.0, SrcQ_IO := 2, SrcQ := 2, Val_Sts := 2, Sts_St1 := 1, Sts_Oper := 1, Sts_Normal := 1, Sts_ExtReqInh := 1, Ack_Fail := 1, Ack_DeviceFault := 1, Ack_IntlkTrip := 1, Ack_IOFault := 1);
   CO2CVMax : REAL := 100.0;
   CO2CVMin : REAL;
   CO2EUMax : REAL := 0.083330005;
   CO2EUMax_Input : REAL := 8.333;
   CO2EUMin : REAL;
   CO2EUMin_Input : REAL;
   CO2ManualSP : REAL := 0.05;
   CO2ManualSP_Input : REAL := 5.0;
   CO2MaxCalc : REAL := 0.083333336;
   CO2PercentOut : REAL := 0.05;
   CO2ProgOper : BOOL := 1;
   conditionedMedia_auto : BOOL := 1;
   ConditionedMedia_Initialize : BOOL := 1;
   ConditionedMedia_PID : PID_ENHANCED := (PV := 10.0, PVEUMax := 300.0, SPOper := 80.0, SPHLimit := 300.0, RatioProg := 1.0, RatioOper := 1.0, RatioHLimit := 1.0, RatioLLimit := 1.0, CVInitReq := 1, CVEUMax := 100.0, CVHLimit := 100.0, PGain := 1.0, IGain := 2.0, PVEDerivative := 1, ProgOperReq := 1, ProgAutoReq := 1, RTSTime := 1, CVInitializing := 1, SP := 80.0, SPPercent := 26.666668, PVPercent := 3.3333335, E := 70.0, EPercent := 23.333334, InitPrimary := 1, Ratio := 1.0, Auto := 1, DeltaT := 1.0);   // DO rich media addition pump
   ConditionedMedia_Scaler : SCALE := (InRawMax := 100.0, InEUMax := 100.0);
   ConditionedMedia_Scaler1 : SCALE := (InRawMax := 100.0, InEUMax := 60.0);
   ConditionedMedia_Scaler2 : SCALE;
   conditionedMediaONS : BOOL := 1;
   conditionedMediaONS2 : BOOL;
   CondMed_AdjustInProgress : BOOL;
   CondMedEUMax : REAL;
   CondMedEUMin : REAL;
   CondMedRawMax : REAL := 100.0;
   CondMedRawMin : REAL;
   Datalog_Trigger : BOOL;   // Toggles Datalogging
   DO_HiDev : REAL;   // hi deviation alarm
   DO_LoDev : REAL;   // low deviation alarm
   DO_ON : BOOL := 1;
   DO_PID_AUTOREQ : BOOL := 1;
   DOpbs : PID_ENHANCED := (PV := 12.0, PVEUMax := 100.0, SPOper := 10.0, SPHLimit := 100.0, RatioProg := 1.0, RatioOper := 1.0, RatioHLimit := 1.0, RatioLLimit := 1.0, CVInitReq := 1, CVOper := 50.0, CVPrevious := 50.0, CVEUMax := 100.0, CVEUMin := -100.0, CVHLimit := 100.0, PGain := 1.0, IGain := 5.0, PVEDerivative := 1, ProgOperReq := 1, RTSTime := 1, CV := 50.0, CVInitializing := 1, SP := 10.0, SPPercent := 10.0, PVPercent := 12.0, E := -2.0, EPercent := -2.0, InitPrimary := 1, Ratio := 1.0, DevHAlarm := 1, Auto := 1, DeltaT := 1.0);
   DOPID_INITIALIZE : BOOL := 1;
   DOtestPV : REAL := 25.0;
   EStop : P_DIn := (Inp_PV := 1, Inp_Target := 1, Inp_Gate := 1, Cfg_NormTextVis := 1, Cfg_HasTgtDisagreeAlm := 1, Cfg_TgtDisagreeAckReqd := 1, Cfg_IOFaultAckReqd := 1, Cfg_TgtDisagreeSeverity := 750, Cfg_IOFaultSeverity := 1000, Set_SimPV := 1, SrcQ_IO := 1, SrcQ := 18, Val_Sts := 7, Val_NotifyAll := 1, Val_UnackAlmC := 1, Sts := 1, Sts_PV := 1, Sts_SubstPV := 1, Sts_MaintByp := 1, Sts_RdyAck := 1, Sts_TgtDisagreeGate := 1, Ack_IOFault := 1);
   FIC110 : P_ValveC := (Inp_IntlkOK := 1, Inp_NBIntlkOK := 1, Cfg_ShedOnIOFault := 1, Cfg_LSFail := 1, Cfg_HasIntlkObj := 1, Cfg_DecPlcs := 2, Cfg_IntlkTripAckReqd := 1, Cfg_ActuatorFaultAckReqd := 1, Cfg_IOFaultAckReqd := 1, Cfg_IntlkTripSeverity := 500, Cfg_ActuatorFaultSeverity := 1000, Cfg_IOFaultSeverity := 1000, Cfg_MaxCV := 2.0, Cfg_CVEUMax := 2.0, Cfg_CVRawMax := 100.0, Cfg_FdbkRawMax := 100.0, Cfg_CycleT := 10.0, Cfg_OpenRate := 1.0, Cfg_CloseRate := 1.0, Cfg_MaxOnT := 5.0, Cfg_MinOnT := 1.0, Cfg_Deadtime := 1.0, Val_CVEUMax := 2.0, SrcQ_IO := 2, SrcQ := 2, Val_Fdbk := 1, Sts_Available := 1, Sts_Prog := 1, Sts_Normal := 1, Sts_ExtReqInh := 1, Ack_IntlkTrip := 1, Ack_ActuatorFault := 1, Ack_IOFault := 1);   // PBS CCA
   FIC110_intlk : P_Intlk := (Cfg_Bypassable := 2#0000_0000_0000_0001, Sts_IntlkOK := 1, Sts_NBIntlkOK := 1, Sts_FirstOut := 2#0000_0000_0000_0001);
   FIC120 : P_ValveC := (Inp_IntlkOK := 1, Inp_NBIntlkOK := 1, Cfg_ShedOnIOFault := 1, Cfg_LSFail := 1, Cfg_HasIntlkObj := 1, Cfg_DecPlcs := 2, Cfg_IntlkTripAckReqd := 1, Cfg_ActuatorFaultAckReqd := 1, Cfg_IOFaultAckReqd := 1, Cfg_IntlkTripSeverity := 500, Cfg_ActuatorFaultSeverity := 1000, Cfg_IOFaultSeverity := 1000, Cfg_MaxCV := 2.0, Cfg_CVEUMax := 2.0, Cfg_CVRawMax := 100.0, Cfg_FdbkRawMax := 100.0, Cfg_CycleT := 10.0, Cfg_OpenRate := 0.2, Cfg_CloseRate := 0.2, Cfg_MaxOnT := 5.0, Cfg_MinOnT := 1.0, Cfg_Deadtime := 1.0, Val_CVEUMax := 2.0, SrcQ_IO := 2, SrcQ := 2, Val_Fdbk := 1, Sts_Available := 1, Sts_Prog := 1, Sts_Normal := 1, Sts_ExtReqInh := 1, Ack_IntlkTrip := 1, Ack_ActuatorFault := 1, Ack_IOFault := 1);   // O2 pbs
   FIC120_intlk : P_Intlk := (Sts_IntlkOK := 1, Sts_NBIntlkOK := 1, Sts_FirstOut := 2#0000_0000_0000_0001);
   FIC130 : P_ValveC := (Inp_IntlkOK := 1, Inp_NBIntlkOK := 1, Cfg_ShedOnIOFault := 1, Cfg_LSFail := 1, Cfg_HasIntlkObj := 1, Cfg_DecPlcs := 2, Cfg_IntlkTripAckReqd := 1, Cfg_ActuatorFaultAckReqd := 1, Cfg_IOFaultAckReqd := 1, Cfg_IntlkTripSeverity := 500, Cfg_ActuatorFaultSeverity := 1000, Cfg_IOFaultSeverity := 1000, Cfg_MaxCV := 0.5, Cfg_CVEUMax := 0.5, Cfg_CVRawMax := 100.0, Cfg_FdbkRawMax := 100.0, Cfg_CycleT := 10.0, Cfg_OpenRate := 0.2, Cfg_CloseRate := 0.2, Cfg_MaxOnT := 5.0, Cfg_MinOnT := 1.0, Cfg_Deadtime := 1.0, Val_CVEUMax := 0.5, SrcQ_IO := 2, SrcQ := 2, Val_Fdbk := 1, Sts_Available := 1, Sts_Prog := 1, Sts_Normal := 1, Sts_ExtReqInh := 1, Ack_IntlkTrip := 1, Ack_ActuatorFault := 1, Ack_IOFault := 1);   // CO2 pbs
   FIC130_intlk : P_Intlk := (Sts_IntlkOK := 1, Sts_NBIntlkOK := 1, Sts_FirstOut := 2#0000_0000_0000_0001);
   FIC140 : P_ValveC := (Inp_IntlkOK := 1, Inp_NBIntlkOK := 1, Cfg_ShedOnIOFault := 1, Cfg_LSFail := 1, Cfg_HasIntlkObj := 1, Cfg_DecPlcs := 2, Cfg_IntlkTripAckReqd := 1, Cfg_ActuatorFaultAckReqd := 1, Cfg_IOFaultAckReqd := 1, Cfg_IntlkTripSeverity := 500, Cfg_ActuatorFaultSeverity := 1000, Cfg_IOFaultSeverity := 1000, Cfg_MaxCV := 2.0, Cfg_CVEUMax := 2.0, Cfg_CVRawMax := 100.0, Cfg_FdbkRawMax := 100.0, Cfg_CycleT := 10.0, Cfg_OpenRate := 1.0, Cfg_CloseRate := 1.0, Cfg_MaxOnT := 5.0, Cfg_MinOnT := 1.0, Cfg_Deadtime := 1.0, XSet_CV := 0.69, Val_CVEUMax := 2.0, SrcQ_IO := 2, SrcQ := 2, Val_Fdbk := 1, Sts_Available := 1, Sts_Prog := 1, Sts_Normal := 1, Sts_ExtReqInh := 1, Ack_IntlkTrip := 1, Ack_ActuatorFault := 1, Ack_IOFault := 1);   // pbs N2 mfc
   FIC140_intlk : P_Intlk := (Sts_IntlkOK := 1, Sts_NBIntlkOK := 1, Sts_FirstOut := 2#0000_0000_0000_0001);
   GasControl_ON : BOOL;
   GasOffOns : BOOL := 1;
   GasOnOns : BOOL;
   Heater_Output : P_AOut := (Inp_NBIntlkOK := 1, Cfg_SetTrack := 1, Cfg_HasIntlkObj := 1, Cfg_ShedOnIOFault := 1, Cfg_DecPlcs := 2, Cfg_IntlkTripAckReqd := 1, Cfg_IOFaultAckReqd := 1, Cfg_IntlkTripSeverity := 500, Cfg_IOFaultSeverity := 1000, Cfg_MaxCV := 20.0, Cfg_CVEUMax := 20.0, Cfg_CVRawMax := 100.0, Val_CVEUMax := 20.0, SrcQ := 20, Sts_NotRdy := 1, Nrdy_Intlk := 1, Sts_Oper := 1, Sts_Normal := 1, Sts_ExtReqInh := 1, Ack_IntlkTrip := 1, Ack_IOFault := 1);   // Heating blanket AO
   Heater_Output_intlk : P_Intlk := (Inp_Intlk00 := 1, Sts_Intlk := 2#0000_0000_0000_0001, Sts_FirstOut := 2#0000_0000_0000_0001);
   Json_Alarm : BOOL;
   KV111 : P_ValveSO := (Inp_PermOK := 1, Inp_NBPermOK := 1, Inp_IntlkOK := 1, Inp_NBIntlkOK := 1, Cfg_LSFail := 1, Cfg_ShedOnFullStall := 1, Cfg_ShedOnTransitStall := 1, Cfg_ShedOnIOFault := 1, Cfg_FullStallAckReqd := 1, Cfg_TransitStallAckReqd := 1, Cfg_IntlkTripAckReqd := 1, Cfg_IOFaultAckReqd := 1, Cfg_FullStallSeverity := 1000, Cfg_TransitStallSeverity := 1000, Cfg_IntlkTripSeverity := 500, Cfg_IOFaultSeverity := 1000, Cfg_SimFdbkT := 2.0, Cfg_FullStallT := 5.0, Cfg_TransitStallT := 10.0, SrcQ_IO := 2, SrcQ := 2, Val_Fdbk := 1, Val_Sts := 1, Sts_Closed := 1, Sts_Oper := 1, Sts_Normal := 1, Sts_ExtReqInh := 1, Ack_FullStall := 1, Ack_TransitStall := 1, Ack_IntlkTrip := 1, Ack_IOFault := 1);   // CCA Overlay Valve
   KV112 : P_ValveSO := (Inp_PermOK := 1, Inp_NBPermOK := 1, Inp_IntlkOK := 1, Inp_NBIntlkOK := 1, Cfg_LSFail := 1, Cfg_ShedOnFullStall := 1, Cfg_ShedOnTransitStall := 1, Cfg_ShedOnIOFault := 1, Cfg_FullStallAckReqd := 1, Cfg_TransitStallAckReqd := 1, Cfg_IntlkTripAckReqd := 1, Cfg_IOFaultAckReqd := 1, Cfg_FullStallSeverity := 1000, Cfg_TransitStallSeverity := 1000, Cfg_IntlkTripSeverity := 500, Cfg_IOFaultSeverity := 1000, Cfg_SimFdbkT := 2.0, Cfg_FullStallT := 5.0, Cfg_TransitStallT := 10.0, SrcQ_IO := 2, SrcQ := 2, Val_Fdbk := 1, Val_Sts := 1, Sts_Closed := 1, Sts_Oper := 1, Sts_Normal := 1, Sts_ExtReqInh := 1, Ack_FullStall := 1, Ack_TransitStall := 1, Ack_IntlkTrip := 1, Ack_IOFault := 1);   // CCA Sparge Valve
   KV121 : P_ValveSO := (Inp_PermOK := 1, Inp_NBPermOK := 1, Inp_IntlkOK := 1, Inp_NBIntlkOK := 1, Cfg_LSFail := 1, Cfg_ShedOnFullStall := 1, Cfg_ShedOnTransitStall := 1, Cfg_ShedOnIOFault := 1, Cfg_FullStallAckReqd := 1, Cfg_TransitStallAckReqd := 1, Cfg_IntlkTripAckReqd := 1, Cfg_IOFaultAckReqd := 1, Cfg_FullStallSeverity := 1000, Cfg_TransitStallSeverity := 1000, Cfg_IntlkTripSeverity := 500, Cfg_IOFaultSeverity := 1000, Cfg_SimFdbkT := 2.0, Cfg_FullStallT := 5.0, Cfg_TransitStallT := 10.0, SrcQ_IO := 2, SrcQ := 2, Val_Fdbk := 1, Val_Sts := 1, Sts_Closed := 1, Sts_Oper := 1, Sts_Normal := 1, Sts_ExtReqInh := 1, Ack_FullStall := 1, Ack_TransitStall := 1, Ack_IntlkTrip := 1, Ack_IOFault := 1);   // O2 Overlay Valve
   KV122 : P_ValveSO := (Inp_PermOK := 1, Inp_NBPermOK := 1, Inp_IntlkOK := 1, Inp_NBIntlkOK := 1, Cfg_LSFail := 1, Cfg_ShedOnFullStall := 1, Cfg_ShedOnTransitStall := 1, Cfg_ShedOnIOFault := 1, Cfg_FullStallAckReqd := 1, Cfg_TransitStallAckReqd := 1, Cfg_IntlkTripAckReqd := 1, Cfg_IOFaultAckReqd := 1, Cfg_FullStallSeverity := 1000, Cfg_TransitStallSeverity := 1000, Cfg_IntlkTripSeverity := 500, Cfg_IOFaultSeverity := 1000, Cfg_SimFdbkT := 2.0, Cfg_FullStallT := 5.0, Cfg_TransitStallT := 10.0, SrcQ_IO := 2, SrcQ := 2, Val_Fdbk := 1, Val_Sts := 1, Sts_Closed := 1, Sts_Oper := 1, Sts_Normal := 1, Sts_ExtReqInh := 1, Ack_FullStall := 1, Ack_TransitStall := 1, Ack_IntlkTrip := 1, Ack_IOFault := 1);   // O2 Sparge Valve
   KV131 : P_ValveSO := (Inp_PermOK := 1, Inp_NBPermOK := 1, Inp_IntlkOK := 1, Inp_NBIntlkOK := 1, Cfg_LSFail := 1, Cfg_ShedOnFullStall := 1, Cfg_ShedOnTransitStall := 1, Cfg_ShedOnIOFault := 1, Cfg_FullStallAckReqd := 1, Cfg_TransitStallAckReqd := 1, Cfg_IntlkTripAckReqd := 1, Cfg_IOFaultAckReqd := 1, Cfg_FullStallSeverity := 1000, Cfg_TransitStallSeverity := 1000, Cfg_IntlkTripSeverity := 500, Cfg_IOFaultSeverity := 1000, Cfg_SimFdbkT := 2.0, Cfg_FullStallT := 5.0, Cfg_TransitStallT := 10.0, SrcQ_IO := 2, SrcQ := 2, Val_Fdbk := 1, Val_Sts := 1, Sts_Closed := 1, Sts_Oper := 1, Sts_Normal := 1, Sts_ExtReqInh := 1, Ack_FullStall := 1, Ack_TransitStall := 1, Ack_IntlkTrip := 1, Ack_IOFault := 1);   // CO2 Overlay Valve
   KV132 : P_ValveSO := (Inp_PermOK := 1, Inp_NBPermOK := 1, Inp_IntlkOK := 1, Inp_NBIntlkOK := 1, Cfg_LSFail := 1, Cfg_ShedOnFullStall := 1, Cfg_ShedOnTransitStall := 1, Cfg_ShedOnIOFault := 1, Cfg_FullStallAckReqd := 1, Cfg_TransitStallAckReqd := 1, Cfg_IntlkTripAckReqd := 1, Cfg_IOFaultAckReqd := 1, Cfg_FullStallSeverity := 1000, Cfg_TransitStallSeverity := 1000, Cfg_IntlkTripSeverity := 500, Cfg_IOFaultSeverity := 1000, Cfg_SimFdbkT := 2.0, Cfg_FullStallT := 5.0, Cfg_TransitStallT := 10.0, SrcQ_IO := 2, SrcQ := 2, Val_Fdbk := 1, Val_Sts := 1, Sts_Closed := 1, Sts_Oper := 1, Sts_Normal := 1, Sts_ExtReqInh := 1, Ack_FullStall := 1, Ack_TransitStall := 1, Ack_IntlkTrip := 1, Ack_IOFault := 1);   // CO2 Sparge Valve
   KV141 : P_ValveSO := (Inp_PermOK := 1, Inp_NBPermOK := 1, Inp_IntlkOK := 1, Inp_NBIntlkOK := 1, Cfg_LSFail := 1, Cfg_ShedOnFullStall := 1, Cfg_ShedOnTransitStall := 1, Cfg_ShedOnIOFault := 1, Cfg_FullStallAckReqd := 1, Cfg_TransitStallAckReqd := 1, Cfg_IntlkTripAckReqd := 1, Cfg_IOFaultAckReqd := 1, Cfg_FullStallSeverity := 1000, Cfg_TransitStallSeverity := 1000, Cfg_IntlkTripSeverity := 500, Cfg_IOFaultSeverity := 1000, Cfg_SimFdbkT := 2.0, Cfg_FullStallT := 5.0, Cfg_TransitStallT := 10.0, SrcQ_IO := 2, SrcQ := 2, Val_Fdbk := 1, Val_Sts := 1, Sts_Closed := 1, Sts_Oper := 1, Sts_Normal := 1, Sts_ExtReqInh := 1, Ack_FullStall := 1, Ack_TransitStall := 1, Ack_IntlkTrip := 1, Ack_IOFault := 1);   // N2 Overlay Valve
   KV142 : P_ValveSO := (Inp_PermOK := 1, Inp_NBPermOK := 1, Inp_IntlkOK := 1, Inp_NBIntlkOK := 1, Cfg_LSFail := 1, Cfg_ShedOnFullStall := 1, Cfg_ShedOnTransitStall := 1, Cfg_ShedOnIOFault := 1, Cfg_FullStallAckReqd := 1, Cfg_TransitStallAckReqd := 1, Cfg_IntlkTripAckReqd := 1, Cfg_IOFaultAckReqd := 1, Cfg_FullStallSeverity := 1000, Cfg_TransitStallSeverity := 1000, Cfg_IntlkTripSeverity := 500, Cfg_IOFaultSeverity := 1000, Cfg_SimFdbkT := 2.0, Cfg_FullStallT := 5.0, Cfg_TransitStallT := 10.0, SrcQ_IO := 2, SrcQ := 2, Val_Fdbk := 1, Val_Sts := 1, Sts_Closed := 1, Sts_Oper := 1, Sts_Normal := 1, Sts_ExtReqInh := 1, Ack_FullStall := 1, Ack_TransitStall := 1, Ack_IntlkTrip := 1, Ack_IOFault := 1);   // N2 Sparge Valve
   Level_Control_Enable : BOOL := 1;
   Level_Deadband_High_SP : REAL := 6.0;
   Level_Deadband_Low_SP : REAL := 4.0;
   LIT801 : P_AInAdv := (Inp_HiHiGate := 1, Inp_HiGate := 1, Inp_LoGate := 1, Inp_LoLoGate := 1, Inp_HiRoCGate := 1, Inp_HiDevGate := 1, Inp_LoDevGate := 1, Inp_FailGate := 1, Cfg_PVDecPlcs := 2, Cfg_HasHiHiAlm := 1, Cfg_HasHiAlm := 1, Cfg_HasLoAlm := 1, Cfg_HasLoLoAlm := 1, Cfg_HiHiAckReqd := 1, Cfg_HiAckReqd := 1, Cfg_LoAckReqd := 1, Cfg_HiRoCAckReqd := 1, Cfg_HiDevAckReqd := 1, Cfg_LoDevAckReqd := 1, Cfg_FailAckReqd := 1, Cfg_HiHiSeverity := 750, Cfg_HiSeverity := 500, Cfg_LoSeverity := 500, Cfg_LoLoSeverity := 750, Cfg_HiRoCSeverity := 500, Cfg_HiDevSeverity := 500, Cfg_LoDevSeverity := 500, Cfg_FailSeverity := 1000, Cfg_InpRawMax := 100.0, Cfg_PVEUMax := 100.0, Cfg_RateTime := 1.0, Cfg_CtrlHiHiLim := 1.5e+38, Cfg_CtrlHiHiDB := 1.0, Cfg_CtrlHiLim := 1.5e+38, Cfg_CtrlHiDB := 1.0, Cfg_CtrlLoLim := -1.5e+38, Cfg_CtrlLoDB := 1.0, Cfg_CtrlLoLoLim := -1.5e+38, Cfg_CtrlLoLoDB := 1.0, Cfg_HiHiLim := 30.0, Cfg_HiHiDB := 1.0, Cfg_HiLim := 1.5e+38, Cfg_HiDB := 1.0, Cfg_LoLim := -1.5e+38, Cfg_LoDB := 1.0, Cfg_LoLoLim := 2.0, Cfg_HiRoCLim := 1.5e+38, Cfg_HiRoCDB := 1.0, Cfg_HiDevLim := 1.5e+38, Cfg_HiDevDB := 1.0, Cfg_LoDevLim := -1.5e+38, Cfg_LoDevDB := 1.0, Cfg_FailHiLim := 103.958336, Cfg_FailLoLim := -2.0833333, Cfg_FailDB := 0.41666666, MSet_SubstPV := 4.3, Val := 4.3, Val_PVMinCapt := 4.3, Val_PVMaxCapt := 4.3, Val_PVEUMax := 100.0,
        SrcQ_IO := 1, SrcQ := 18, Sts_SubstPV := 1, Sts_MaintByp := 1, Sts_HiHiGate := 1, Ack_HiHi := 1, Sts_HiGate := 1, Ack_Hi := 1, Sts_LoGate := 1, Ack_Lo := 1, Sts_LoLoGate := 1, Ack_LoLo := 1, Sts_HiRoCGate := 1, Ack_HiRoC := 1, Sts_HiDevGate := 1, Ack_HiDev := 1, Sts_LoDevGate := 1, Ack_LoDev := 1, Sts_FailGate := 1, Ack_Fail := 1);   // Level Value From BRX
   ManualDO_CV : REAL := 50.0;
   ManualpH_CV : REAL;
   MCV_FillWeight : REAL := 15.0;
   MCV_HiAdj : BOOL;   // MCV hi adjust active
   MCV_HiAdjEnable : BOOL := 1;
   MCV_HiAdjTimer : TIMER := (PRE := 20000);
   MCV_HiAdjTimeSP : REAL := 20.0;
   MCV_HiSP : REAL := 15.0;
   MCV_InitialFill : BOOL;
   MCV_InitialFillRunning : BOOL;
   MCV_InitialFillSpeed : REAL := 100.0;
   MCV_LoAdjTimer : TIMER := (PRE := 10000);
   MCV_LoSP : REAL := 16.0;
   MCV_LoTimerSP : REAL := 10.0;
   MediaAdj_InProgress : BOOL;
   MediaFill_ON : BOOL;
   MediaLoSpeed : REAL := 50.0;
   N2_3way : P_D4SD := (Inp_PermOK0 := 1, Inp_NBPermOK0 := 1, Inp_PermOK1 := 1, Inp_NBPermOK1 := 1, Inp_PermOK2 := 1, Inp_NBPermOK2 := 1, Inp_PermOK3 := 1, Inp_NBPermOK3 := 1, Inp_IntlkOK := 1, Inp_NBIntlkOK := 1, Cfg_NumStates := 2, Cfg_OutSt0Write := 2#0000_1111, Cfg_OutSt0State := 2#0000_0001, Cfg_OutSt1Write := 2#0000_1111, Cfg_OutSt1State := 2#0000_0010, Cfg_OutSt2Write := 2#0000_1111, Cfg_OutSt2State := 2#0000_0100, Cfg_OutSt3Write := 2#0000_1111, Cfg_OutSt3State := 2#0000_1000, Cfg_FdbkSt0State := 2#0000_0001, Cfg_FdbkSt1State := 2#0000_0010, Cfg_FdbkSt2State := 2#0000_0100, Cfg_FdbkSt3State := 2#0000_1000, Cfg_FailAckReqd := 1, Cfg_DeviceFaultAckReqd := 1, Cfg_IntlkTripAckReqd := 1, Cfg_IOFaultAckReqd := 1, Cfg_FailSeverity := 1000, Cfg_DeviceFaultSeverity := 1000, Cfg_IntlkTripSeverity := 500, Cfg_IOFaultSeverity := 1000, Cfg_SimFdbkT := 2.0, Cfg_FailT := 10.0, SrcQ_IO := 2, SrcQ := 2, Val_Sts := 1, Sts_St0 := 1, Sts_Oper := 1, Sts_Normal := 1, Sts_ExtReqInh := 1, Ack_Fail := 1, Ack_DeviceFault := 1, Ack_IntlkTrip := 1, Ack_IOFault := 1);
   N2CVMax : REAL := -5.0;
   N2CVMin : REAL := -100.0;
   N2EUMax : REAL;
   N2EUMax_Input : REAL;
   N2EUMin : REAL := 0.33333;
   N2EUMin_Input : REAL := 33.333;
   N2ManualSP : REAL;
   N2ManualSP_Input : REAL;
   N2MaxCalc : REAL := 0.33333334;
   N2PercentOut : REAL;
   N2ProgOper : BOOL;
   N2Scaler : SCALE := (InRawMax := -5.0, InRawMin := -100.0, InEUMin := 0.33333, Limiting := 1, MaxAlarm := 1);
   O2_3way : P_D4SD := (Inp_PermOK0 := 1, Inp_NBPermOK0 := 1, Inp_PermOK1 := 1, Inp_NBPermOK1 := 1, Inp_PermOK2 := 1, Inp_NBPermOK2 := 1, Inp_PermOK3 := 1, Inp_NBPermOK3 := 1, Inp_IntlkOK := 1, Inp_NBIntlkOK := 1, Cfg_NumStates := 2, Cfg_OutSt0Write := 2#0000_1111, Cfg_OutSt0State := 2#0000_0001, Cfg_OutSt1Write := 2#0000_1111, Cfg_OutSt1State := 2#0000_0010, Cfg_OutSt2Write := 2#0000_1111, Cfg_OutSt2State := 2#0000_0100, Cfg_OutSt3Write := 2#0000_1111, Cfg_OutSt3State := 2#0000_1000, Cfg_FdbkSt0State := 2#0000_0001, Cfg_FdbkSt1State := 2#0000_0010, Cfg_FdbkSt2State := 2#0000_0100, Cfg_FdbkSt3State := 2#0000_1000, Cfg_FailAckReqd := 1, Cfg_DeviceFaultAckReqd := 1, Cfg_IntlkTripAckReqd := 1, Cfg_IOFaultAckReqd := 1, Cfg_FailSeverity := 1000, Cfg_DeviceFaultSeverity := 1000, Cfg_IntlkTripSeverity := 500, Cfg_IOFaultSeverity := 1000, Cfg_SimFdbkT := 2.0, Cfg_FailT := 10.0, SrcQ_IO := 2, SrcQ := 2, Val_Sts := 2, Sts_St1 := 1, Sts_Oper := 1, Sts_Normal := 1, Sts_ExtReqInh := 1, Ack_Fail := 1, Ack_DeviceFault := 1, Ack_IntlkTrip := 1, Ack_IOFault := 1);
   O2CVMax : REAL := 100.0;
   O2CVMin : REAL := 5.0;
   O2EUMax : REAL := 0.33333;
   O2EUMax_Input : REAL := 33.333;
   O2EUMin : REAL;
   O2EUMin_Input : REAL;
   O2ManualSP : REAL;
   O2ManualSP_Input : REAL;
   O2MaxCalc : REAL := 0.33333334;
   O2PercentOut : REAL;
   O2ProgOper : BOOL;
   O2Scaler : SCALE := (InRawMax := 100.0, InRawMin := 5.0, InEUMax := 0.33333, Limiting := 1, MinAlarm := 1);
   ONS : DINT[3];
   P101 : P_VSD := (Inp_Ready := 1, Inp_CommandDir := 1, Inp_ActualDir := 1, Inp_FwdPermOK := 1, Inp_FwdNBPermOK := 1, Inp_RevPermOK := 1, Inp_RevNBPermOK := 1, Inp_IntlkOK := 1, Inp_NBIntlkOK := 1, Cfg_HasIntlkObj := 1, Cfg_SetTrack := 1, Cfg_ShedOnFailToStart := 1, Cfg_ShedOnIOFault := 1, Cfg_DecPlcs := 2, Cfg_InpDLDecPlcs := 2, Cfg_OutDLDecPlcs := 2, Cfg_FailToStartAckReqd := 1, Cfg_FailToStopAckReqd := 1, Cfg_IntlkTripAckReqd := 1, Cfg_DriveFaultAckReqd := 1, Cfg_IOFaultAckReqd := 1, Cfg_FailToStartSeverity := 1000, Cfg_FailToStopSeverity := 1000, Cfg_IntlkTripSeverity := 500, Cfg_DriveFaultSeverity := 1000, Cfg_IOFaultSeverity := 1000, Cfg_MaxSpdRef := 400.0, Cfg_SpeedRefRawMax := 32767.0, Cfg_SpeedRefEUMax := 400.0, Cfg_SpeedFdbkRawMax := 32767.0, Cfg_SpeedFdbkEUMax := 400.0, Cfg_InpDatalinkRawMax := 4095.0, Cfg_InpDatalinkEUMax := 409.5, Cfg_OutDatalinkMax := 100.0, Cfg_OutDatalinkRawMax := 4095.0, Cfg_OutDatalinkEUMax := 409.5, Cfg_SimRampT := 10.0, Cfg_FailToStartT := 15.0, Cfg_FailToStopT := 15.0, Cfg_ResetPulseT := 2.0, XSet_SpeedRef := 50.0, Out_SpeedRef := 4095.875, Out_Fwd := 1, Val_SpeedRef := 50.0, Val_SpeedRefEUMax := 400.0, Val_SpeedFdbkEUMax := 400.0, SrcQ_IO := 2, SrcQ := 2, Val_Sts := 1, Sts_Stopped := 1, Sts_CommandDir := 1, Sts_ActualDir := 1, Sts_Oper := 1, Sts_Normal := 1, Sts_ExtReqInh := 1, Ack_FailToStart := 1, Ack_FailToStop := 1, Ack_IntlkTrip := 1, Ack_DriveFault := 1, Ack_IOFault := 1);   // Feed Pump
   P101_Alarm_Reset : AMP_Alarm_Reset := (RPI := 100, Sent := 1, Done := 1, State := 70);
   P101_Cal : Pump_Cal := (Cal_CollectedQuantity := 130.0, Cal_Duration := 0.5, Cal_PumpSpeed := 100.0, Cal_Complete := 1, Cal_EUMax := 260.0);
   P101_Cal_Abort : BOOL;
   P101_Cal_Accept : BOOL;
   P101_Cal_ColConst : REAL := 2.0;
   P101_Cal_Collected : REAL := 100.0;
   P101_Cal_Complete : BOOL := 1;
   P101_Cal_Constant : REAL := 2.0;
   P101_Cal_Max_Flow : REAL := 400.0;
   P101_Cal_Running : BOOL;
   P101_Cal_Speed : REAL := 52.0;   // ml/min
   p101_Cal_Start : BOOL;
   P101_Cal_Steps : REAL := 50.0;
   P101_CalRevs : REAL := 50.0;
   P101_Crash_Stop : AMP_Crash_Stop := (RPI := 100, Sent := 1, Done := 1, State := 70);
   P101_Dose_Abort : BOOL;
   P101_Dose_mL : REAL := 100.0;
   P101_Dose_Running : BOOL;
   P101_Dose_Speed_mlmin : REAL := 200.0;
   P101_Dose_Start : BOOL;
   P101_Enable : AMP_Motor_Enable := (RPI := 100, Sent := 1, Done := 1, State := 70);
   P101_FaultCodeList : P_DescList[1];
   P101_Input_Assembly : AMP_Input_Assembly_v2 := (Status_Code := 9, Voltage := 243, Temp := 490, Main_Board_Inputs := 255, Word11 := 15);
   P101_Input_Assembly_Instance : AMP_Input_Assembly := (Status_Code := 16#0000_0009, Voltage := 24.3, Temp := 49.0, Main_Board_Inputs := 16#00ff);
   P101_intlk : P_Intlk := (Sts_IntlkOK := 1, Sts_NBIntlkOK := 1, Sts_FirstOut := 2#0000_0000_0000_0100);
   P101_Jog_Move : AMP_Jog_Move := (RPI := 100, Start := 1, Speed := 0.41666666, Acc := 2.0, Dec := 2.0, Sent := 1, In_Progress := 1, State := 60);
   P101_MaxRPM : REAL := 200.0;
   P101_Motor_Constant : DINT := 50;
   P101_Relative_Move : AMP_Relative_Move := (RPI := 100, Distance := 50, Speed := 1.6666666, Acc := 3.0, Dec := 3.0, Sent := 1, Done := 1, State := 70);
   P101_Speed : REAL := 50.0;
   P101_Status_Code : AMP_Status_Code := (Input := 16#0000_0009, Motor_Enabled := 1, In_Position := 1);
   P101_Timer : TIMER;
   P101_Update_Jog_Speed : AMP_Update_Jog_Speed := (RPI := 100, Speed := 0.41666666, Sent := 1, In_Progress := 1, State := 60);
   P101Fault : BOOL;
   P101Fault_Output : BOOL;
   P102 : P_VSD := (Inp_Ready := 1, Inp_CommandDir := 1, Inp_ActualDir := 1, Inp_FwdPermOK := 1, Inp_FwdNBPermOK := 1, Inp_RevPermOK := 1, Inp_RevNBPermOK := 1, Inp_IntlkOK := 1, Inp_NBIntlkOK := 1, Cfg_HasIntlkObj := 1, Cfg_SetTrack := 1, Cfg_ShedOnFailToStart := 1, Cfg_ShedOnIOFault := 1, Cfg_DecPlcs := 2, Cfg_InpDLDecPlcs := 2, Cfg_OutDLDecPlcs := 2, Cfg_FailToStartAckReqd := 1, Cfg_FailToStopAckReqd := 1, Cfg_IntlkTripAckReqd := 1, Cfg_DriveFaultAckReqd := 1, Cfg_IOFaultAckReqd := 1, Cfg_FailToStartSeverity := 1000, Cfg_FailToStopSeverity := 1000, Cfg_IntlkTripSeverity := 500, Cfg_DriveFaultSeverity := 1000, Cfg_IOFaultSeverity := 1000, Cfg_MaxSpdRef := 250.0, Cfg_SpeedRefRawMax := 32767.0, Cfg_SpeedRefEUMax := 100.0, Cfg_SpeedFdbkRawMax := 32767.0, Cfg_SpeedFdbkEUMax := 100.0, Cfg_InpDatalinkRawMax := 4095.0, Cfg_InpDatalinkEUMax := 409.5, Cfg_OutDatalinkMax := 100.0, Cfg_OutDatalinkRawMax := 4095.0, Cfg_OutDatalinkEUMax := 409.5, Cfg_SimRampT := 10.0, Cfg_FailToStartT := 15.0, Cfg_FailToStopT := 15.0, Cfg_ResetPulseT := 2.0, XSet_SpeedRef := 200.0, Out_SpeedRef := 65534.0, Out_Fwd := 1, Val_SpeedRef := 200.0, Val_SpeedRefEUMax := 100.0, Val_SpeedFdbkEUMax := 100.0, SrcQ_IO := 2, SrcQ := 2, Val_Sts := 1, Sts_Stopped := 1, Sts_CommandDir := 1, Sts_ActualDir := 1, Sts_Oper := 1, Sts_Normal := 1, Sts_ExtReqInh := 1, Ack_FailToStart := 1, Ack_FailToStop := 1, Ack_IntlkTrip := 1, Ack_DriveFault := 1, Ack_IOFault := 1);   // Media Pump
   P102_Alarm_Reset : AMP_Alarm_Reset := (RPI := 100, Sent := 1, Done := 1, State := 70);
   P102_Cal : Pump_Cal := (Cal_Duration := 0.5, Cal_PumpSpeed := 100.0, Cal_Aborted := 1);
   P102_Cal_Abort : BOOL;
   P102_Cal_Accept : BOOL;
   P102_Cal_ColConst : REAL := 1.e-04;
   P102_Cal_Collected : REAL := 100.0;
   P102_Cal_Complete : BOOL;
   P102_Cal_Constant : REAL;
   P102_Cal_Max_Flow : REAL;
   P102_Cal_Running : BOOL;
   P102_Cal_Speed : REAL;   // ml/min
   P102_Cal_Steps : REAL;
   P102_CalRevs : REAL;
   P102_Crash_Stop : AMP_Crash_Stop := (RPI := 100, In_Progress := 1, Error := 1, State := 10);
   P102_Dose_Abort : BOOL;
   P102_Dose_mL : REAL;
   P102_Dose_Running : BOOL;
   P102_Dose_Speed_mlmin : REAL;
   P102_Dose_Start : BOOL;
   P102_Enable : AMP_Motor_Enable := (RPI := 100, Sent := 1, In_Progress := 1, State := 60);
   P102_FaultCodeList : P_DescList[1];
   P102_Input_Assembly : AMP_Input_Assembly_v2;
   P102_Input_Assembly_Instance : AMP_Input_Assembly;
   P102_intlk : P_Intlk := (Sts_IntlkOK := 1, Sts_NBIntlkOK := 1, Sts_FirstOut := 2#0000_0000_0000_0100);
   P102_Jog_Move : AMP_Jog_Move := (RPI := 100, Start := 1, Speed := inf, Sent := 1, In_Progress := 1, State := 60);
   P102_MaxRPM : REAL;
   P102_Motor_Constant : REAL;
   P102_Motor_Enable : AMP_Motor_Enable := (RPI := 100, State := 10);
   P102_Relative_Move : AMP_Relative_Move := (RPI := 100, Error := 1, State := 10);
   P102_Status_Code : AMP_Status_Code;
   P102_Update_Jog_Speed : AMP_Update_Jog_Speed := (RPI := 100, Speed := inf, Sent := 1, In_Progress := 1, State := 60);
   P103 : P_VSD := (Inp_Ready := 1, Inp_CommandDir := 1, Inp_ActualDir := 1, Inp_FwdPermOK := 1, Inp_FwdNBPermOK := 1, Inp_RevPermOK := 1, Inp_RevNBPermOK := 1, Inp_IntlkOK := 1, Inp_NBIntlkOK := 1, Cfg_HasIntlkObj := 1, Cfg_SetTrack := 1, Cfg_ShedOnFailToStart := 1, Cfg_ShedOnIOFault := 1, Cfg_DecPlcs := 2, Cfg_InpDLDecPlcs := 2, Cfg_OutDLDecPlcs := 2, Cfg_FailToStartAckReqd := 1, Cfg_FailToStopAckReqd := 1, Cfg_IntlkTripAckReqd := 1, Cfg_DriveFaultAckReqd := 1, Cfg_IOFaultAckReqd := 1, Cfg_FailToStartSeverity := 1000, Cfg_FailToStopSeverity := 1000, Cfg_IntlkTripSeverity := 500, Cfg_DriveFaultSeverity := 1000, Cfg_IOFaultSeverity := 1000, Cfg_MaxSpdRef := 100.0, Cfg_SpeedRefRawMax := 32767.0, Cfg_SpeedRefEUMax := 100.0, Cfg_SpeedFdbkRawMax := 32767.0, Cfg_SpeedFdbkEUMax := 100.0, Cfg_InpDatalinkRawMax := 4095.0, Cfg_InpDatalinkEUMax := 409.5, Cfg_OutDatalinkMax := 100.0, Cfg_OutDatalinkRawMax := 4095.0, Cfg_OutDatalinkEUMax := 409.5, Cfg_SimRampT := 10.0, Cfg_FailToStartT := 15.0, Cfg_FailToStopT := 15.0, Cfg_ResetPulseT := 2.0, XSet_SpeedRef := 30.0, Out_SpeedRef := 9830.1, Out_Fwd := 1, Val_SpeedRef := 30.0, Val_SpeedRefEUMax := 100.0, Val_SpeedFdbkEUMax := 100.0, SrcQ_IO := 2, SrcQ := 2, Val_Sts := 1, Sts_Stopped := 1, Sts_CommandDir := 1, Sts_ActualDir := 1, Sts_Oper := 1, Sts_Normal := 1, Sts_ExtReqInh := 1, Ack_FailToStart := 1, Ack_FailToStop := 1, Ack_IntlkTrip := 1, Ack_DriveFault := 1, Ack_IOFault := 1);   // Conditioned Media Addition Pump
   P103_Alarm_Reset : AMP_Alarm_Reset := (RPI := 100, Sent := 1, Done := 1, State := 70);
   P103_Cal : Pump_Cal := (Cal_CollectedQuantity := 50.0, Cal_Duration := 0.5, Cal_PumpSpeed := 100.0, Cal_Complete := 1, Cal_EUMax := 100.0);
   P103_Cal_Abort : BOOL;
   P103_Cal_Accept : BOOL;
   P103_Cal_ColConst : REAL;
   P103_Cal_Collected : REAL;
   P103_Cal_Complete : BOOL;
   P103_Cal_Constant : REAL;
   P103_Cal_Max_Flow : REAL;
   P103_Cal_Running : BOOL;
   P103_Cal_Speed : REAL;   // ml/min
   P103_Cal_Steps : REAL;
   P103_CalRevs : REAL;
   P103_Crash_Stop : AMP_Crash_Stop := (RPI := 100, In_Progress := 1, Error := 1, State := 10);
   P103_Dose_Abort : BOOL;
   P103_Dose_mL : REAL;
   P103_Dose_Running : BOOL;
   P103_Dose_Speed_mlmin : REAL;
   P103_Dose_Start : BOOL;
   P103_Enable : AMP_Motor_Enable := (RPI := 100, Sent := 1, In_Progress := 1, State := 60);
   P103_FaultCodeList : P_DescList[1];
   P103_Input_Assembly : AMP_Input_Assembly_v2;
   P103_Input_Assembly_Instance : AMP_Input_Assembly;
   P103_intlk : P_Intlk := (Sts_IntlkOK := 1, Sts_NBIntlkOK := 1, Sts_FirstOut := 2#0000_0000_0000_0100);
   P103_Jog_Move : AMP_Jog_Move := (RPI := 100, Start := 1, Speed := inf, Sent := 1, In_Progress := 1, State := 60);
   P103_MaxRPM : REAL;
   P103_Motor_Constant : REAL;
   P103_Motor_Enable : AMP_Motor_Enable := (RPI := 100, State := 10);
   P103_Relative_Move : AMP_Relative_Move := (RPI := 100, Error := 1, State := 10);
   P103_Status_Code : AMP_Status_Code;
   P103_Update_Jog_Speed : AMP_Update_Jog_Speed := (RPI := 100, Speed := inf, Error := 1, State := 10);
   P104 : P_VSD := (Inp_Ready := 1, Inp_CommandDir := 1, Inp_ActualDir := 1, Inp_FwdPermOK := 1, Inp_FwdNBPermOK := 1, Inp_RevPermOK := 1, Inp_RevNBPermOK := 1, Inp_IntlkOK := 1, Inp_NBIntlkOK := 1, Cfg_HasReverse := 1, Cfg_HasIntlkObj := 1, Cfg_SetTrack := 1, Cfg_ShedOnFailToStart := 1, Cfg_ShedOnIOFault := 1, Cfg_DecPlcs := 2, Cfg_InpDLDecPlcs := 2, Cfg_OutDLDecPlcs := 2, Cfg_FailToStartAckReqd := 1, Cfg_FailToStopAckReqd := 1, Cfg_IntlkTripAckReqd := 1, Cfg_DriveFaultAckReqd := 1, Cfg_IOFaultAckReqd := 1, Cfg_FailToStartSeverity := 1000, Cfg_FailToStopSeverity := 1000, Cfg_IntlkTripSeverity := 500, Cfg_DriveFaultSeverity := 1000, Cfg_IOFaultSeverity := 1000, Cfg_MaxSpdRef := 100.0, Cfg_SpeedRefRawMax := 32767.0, Cfg_SpeedRefEUMax := 220.0, Cfg_SpeedFdbkRawMax := 32767.0, Cfg_SpeedFdbkEUMax := 220.0, Cfg_InpDatalinkRawMax := 4095.0, Cfg_InpDatalinkEUMax := 409.5, Cfg_OutDatalinkMax := 100.0, Cfg_OutDatalinkRawMax := 4095.0, Cfg_OutDatalinkEUMax := 409.5, Cfg_SimRampT := 10.0, Cfg_FailToStartT := 15.0, Cfg_FailToStopT := 15.0, Cfg_ResetPulseT := 2.0, XSet_SpeedRef := 52.0, Out_SpeedRef := 7744.9272, Out_Fwd := 1, Val_SpeedRef := 52.0, Val_SpeedRefEUMax := 220.0, Val_SpeedFdbkEUMax := 220.0, SrcQ_IO := 2, SrcQ := 2, Val_Sts := 1, Sts_Stopped := 1, Sts_CommandDir := 1, Sts_ActualDir := 1, Sts_Oper := 1, Sts_Normal := 1, Sts_ExtReqInh := 1, Ack_FailToStart := 1, Ack_FailToStop := 1, Ack_IntlkTrip := 1, Ack_DriveFault := 1,
        Ack_IOFault := 1);   // Recirculation Pump
   P104_Alarm_Reset : AMP_Alarm_Reset := (RPI := 100, Sent := 1, Done := 1, State := 70);
   P104_Cal : Pump_Cal := (Cal_CollectedQuantity := 110.0, Cal_Duration := 0.5, Cal_PumpSpeed := 100.0, Cal_Complete := 1, Cal_EUMax := 220.0);
   P104_Cal_Abort : BOOL;
   P104_Cal_Accept : BOOL;
   P104_Cal_ColConst : REAL;
   P104_Cal_Collected : REAL;
   P104_Cal_Complete : BOOL;
   P104_Cal_Constant : REAL;
   P104_Cal_Max_Flow : REAL;
   P104_Cal_Running : BOOL;
   P104_Cal_Speed : REAL;   // ml/min
   P104_Cal_Steps : REAL;
   P104_CalRevs : REAL;
   P104_Crash_Stop : AMP_Crash_Stop := (RPI := 100, In_Progress := 1, Error := 1, State := 10);
   P104_Dose_Abort : BOOL;
   P104_Dose_mL : REAL;
   P104_Dose_Running : BOOL;
   P104_Dose_Speed_mlmin : REAL;
   P104_Dose_Start : BOOL;
   P104_Enable : AMP_Motor_Enable := (RPI := 100, Sent := 1, In_Progress := 1, State := 60);
   P104_FaultCodeList : P_DescList[1];
   P104_Input_Assembly : AMP_Input_Assembly_v2;
   P104_Input_Assembly_Instance : AMP_Input_Assembly;
   p104_intlk : P_Intlk := (Sts_IntlkOK := 1, Sts_NBIntlkOK := 1, Sts_FirstOut := 2#0000_0000_0000_0100);
   P104_Jog_Move : AMP_Jog_Move := (RPI := 100, Start := 1, Speed := inf, Sent := 1, In_Progress := 1, State := 60);
   P104_MaxRPM : REAL;
   P104_Motor_Constant : REAL;
   P104_Motor_Enable : AMP_Motor_Enable := (RPI := 100, State := 10);
   P104_Relative_Move : AMP_Relative_Move := (RPI := 100, Error := 1, State := 10);
   P104_Status_Code : AMP_Status_Code;
   P104_Update_Jog_Speed : AMP_Update_Jog_Speed := (RPI := 100, Speed := inf, Sent := 1, In_Progress := 1, State := 60);
   P105 : P_VSD := (Inp_Ready := 1, Inp_CommandDir := 1, Inp_ActualDir := 1, Inp_FwdPermOK := 1, Inp_FwdNBPermOK := 1, Inp_RevPermOK := 1, Inp_RevNBPermOK := 1, Inp_IntlkOK := 1, Inp_NBIntlkOK := 1, Cfg_HasIntlkObj := 1, Cfg_SetTrack := 1, Cfg_ShedOnFailToStart := 1, Cfg_ShedOnIOFault := 1, Cfg_DecPlcs := 2, Cfg_InpDLDecPlcs := 2, Cfg_OutDLDecPlcs := 2, Cfg_FailToStartAckReqd := 1, Cfg_FailToStopAckReqd := 1, Cfg_IntlkTripAckReqd := 1, Cfg_DriveFaultAckReqd := 1, Cfg_IOFaultAckReqd := 1, Cfg_FailToStartSeverity := 1000, Cfg_FailToStopSeverity := 1000, Cfg_IntlkTripSeverity := 500, Cfg_DriveFaultSeverity := 1000, Cfg_IOFaultSeverity := 1000, Cfg_MaxSpdRef := 60.0, Cfg_SpeedRefRawMax := 32767.0, Cfg_SpeedRefEUMax := 130.0, Cfg_SpeedFdbkRawMax := 32767.0, Cfg_SpeedFdbkEUMax := 130.0, Cfg_InpDatalinkRawMax := 4095.0, Cfg_InpDatalinkEUMax := 409.5, Cfg_OutDatalinkMax := 100.0, Cfg_OutDatalinkRawMax := 4095.0, Cfg_OutDatalinkEUMax := 409.5, Cfg_SimRampT := 10.0, Cfg_FailToStartT := 15.0, Cfg_FailToStopT := 15.0, Cfg_ResetPulseT := 2.0, XSet_SpeedRef := 50.0, Out_SpeedRef := 12602.692, Out_Fwd := 1, Val_SpeedRef := 50.0, Val_SpeedRefEUMax := 130.0, Val_SpeedFdbkEUMax := 130.0, SrcQ_IO := 2, SrcQ := 2, Val_Sts := 1, Sts_Stopped := 1, Sts_CommandDir := 1, Sts_ActualDir := 1, Sts_Oper := 1, Sts_Normal := 1, Sts_ExtReqInh := 1, Ack_FailToStart := 1, Ack_FailToStop := 1, Ack_IntlkTrip := 1, Ack_DriveFault := 1, Ack_IOFault := 1);   // Spent Media Pump
   P105_Abort : BOOL;
   P105_Cal : Pump_Cal;
   P105_Cal_Abort : BOOL;
   P105_Cal_Accept : BOOL;
   P105_Cal_ColConst : REAL;
   P105_Cal_Collected : REAL;
   P105_Cal_Complete : BOOL;
   P105_Cal_Constant : REAL;
   P105_Cal_Max_Flow : REAL;
   P105_Cal_Running : BOOL;
   P105_Cal_Speed : REAL;
   P105_Cal_Steps : REAL;
   P105_CalRevs : REAL;
   P105_Crash_Stop : AMP_Crash_Stop := (RPI := 100, State := 10);
   P105_DeciRPM : REAL := 200.0;
   P105_Dose : REAL := 100.0;   // mL
   P105_Dose_Running : BOOL;
   P105_DoseSpeed : REAL := 200.0;   // mL/min
   P105_FaultCodeList : P_DescList[1];
   P105_intlk : P_Intlk := (Sts_IntlkOK := 1, Sts_NBIntlkOK := 1, Sts_FirstOut := 2#0000_0000_0000_0100);
   P105_MaxRPM : REAL;
   P105_mLrev : REAL := 10.0;   // mL/rev
   P105_Motor_Constant : REAL;
   P105_Relative_Move : AMP_Relative_Move := (RPI := 100, State := 10);
   P105_StartDose : BOOL;
   P105_Timer : TIMER := (PRE := 30000);
   Perfusion_Level_Aggression : REAL := 10.0;
   Perfusion_Off : BOOL;
   Perfusion_On : BOOL;
   pH_HiDev : REAL;   // ph hi deviation
   pH_Initialize : BOOL := 1;
   pH_LoDev : REAL;   // pH Lo deviation alarm
   PH_On : BOOL := 1;
   pH_PID_AUTOREQ : BOOL := 1;
   PHpbs : PID_ENHANCED := (PV := 7.2, PVEUMax := 14.0, SPProg := 7.0, SPOper := 10.0, SPHLimit := 14.0, RatioProg := 1.0, RatioOper := 1.0, RatioHLimit := 1.0, RatioLLimit := 1.0, CVInitReq := 1, CVEUMax := 100.0, CVHLimit := 100.0, PGain := 1.0, IGain := 5.0, PVEDerivative := 1, ProgOperReq := 1, RTSTime := 1, CVInitializing := 1, SP := 10.0, SPPercent := 71.42857, PVPercent := 51.42857, E := 2.8000002, EPercent := 20.000004, InitPrimary := 1, Ratio := 1.0, DevLAlarm := 1, Auto := 1, DeltaT := 1.0);
   pHtestPV : REAL;
   PlaceHolderFeedback1 : REAL;
   PlaceHolderFeedback2 : REAL;
   PlaceHolderFeedback3 : REAL;
   PlaceHolderFeedback4 : REAL;
   PlaceHolderIOFault : DINT[3];
   PlaceHolderOutput1 : REAL;
   PlaceHolderOutput2 : REAL;
   PlaceHolderOutput3 : REAL;
   PlaceHolderOutput4 : REAL;
   REAL : DINT;
   Recirc_HiSP1 : REAL := 1.1;   // BRX Hi recirc hi speed modifier
   Recirc_LoSP1 : REAL := 0.8;   // MCV Hi recirc lo speed modifier
   Recirc_LoSP2 : REAL := 0.9;   // BRX Lo recirc lo speed modifier
   SIC401 : P_VSD := (Inp_Ready := 1, Inp_CommandDir := 1, Inp_ActualDir := 1, Inp_FwdPermOK := 1, Inp_FwdNBPermOK := 1, Inp_RevPermOK := 1, Inp_RevNBPermOK := 1, Inp_IntlkOK := 1, Inp_NBIntlkOK := 1, Cfg_HasIntlkObj := 1, Cfg_SetTrack := 1, Cfg_ShedOnFailToStart := 1, Cfg_ShedOnIOFault := 1, Cfg_DecPlcs := 2, Cfg_InpDLDecPlcs := 2, Cfg_OutDLDecPlcs := 2, Cfg_FailToStartAckReqd := 1, Cfg_FailToStopAckReqd := 1, Cfg_IntlkTripAckReqd := 1, Cfg_DriveFaultAckReqd := 1, Cfg_IOFaultAckReqd := 1, Cfg_FailToStartSeverity := 1000, Cfg_FailToStopSeverity := 1000, Cfg_IntlkTripSeverity := 500, Cfg_DriveFaultSeverity := 1000, Cfg_IOFaultSeverity := 1000, Cfg_MaxSpdRef := 60.0, Cfg_SpeedRefRawMax := 32767.0, Cfg_SpeedRefEUMax := 130.0, Cfg_SpeedFdbkRawMax := 32767.0, Cfg_SpeedFdbkEUMax := 130.0, Cfg_InpDatalinkRawMax := 4095.0, Cfg_InpDatalinkEUMax := 409.5, Cfg_OutDatalinkMax := 100.0, Cfg_OutDatalinkRawMax := 4095.0, Cfg_OutDatalinkEUMax := 409.5, Cfg_SimRampT := 10.0, Cfg_FailToStartT := 15.0, Cfg_FailToStopT := 15.0, Cfg_ResetPulseT := 2.0, PSet_SpeedRef := 20.0, XSet_SpeedRef := 20.0, Out_SpeedRef := 5041.077, Out_Fwd := 1, Val_SpeedRef := 20.0, Val_SpeedRefEUMax := 130.0, Val_SpeedFdbkEUMax := 130.0, SrcQ_IO := 2, SrcQ := 2, Val_Sts := 1, Sts_Stopped := 1, Sts_CommandDir := 1, Sts_ActualDir := 1, Sts_Oper := 1, Sts_Normal := 1, Sts_ExtReqInh := 1, Ack_FailToStart := 1, Ack_FailToStop := 1, Ack_IntlkTrip := 1, Ack_DriveFault := 1,
        Ack_IOFault := 1);   // Agitator
   SIC401_FaultCodeList : P_DescList[1];   // made for agaitor p_VSD block
   SIC401_intlk : P_Intlk := (Sts_IntlkOK := 1, Sts_NBIntlkOK := 1, Sts_FirstOut := 2#0000_0000_0000_0010);
   Temp_Control_On : BOOL := 1;   // Temp On HMI Button
   Temp_Initialize : BOOL := 1;
   Temp_Limit_Adm : REAL := 20.0;
   Temp_OutputLimit : REAL := 20.0;
   Temp_PID : PID_ENHANCED := (PV := 95.0, PVEUMax := 100.0, SPOper := 10.0, SPHLimit := 100.0, RatioProg := 1.0, RatioOper := 1.0, RatioHLimit := 1.0, RatioLLimit := 1.0, CVInitReq := 1, CVEUMax := 100.0, CVHLimit := 100.0, PGain := 10.0, IGain := 5.0, PVEDerivative := 1, ProgOperReq := 1, ProgAutoReq := 1, RTSTime := 1, CVInitializing := 1, SP := 10.0, SPPercent := 10.0, PVPercent := 95.0, E := -85.0, EPercent := -85.0, InitPrimary := 1, Ratio := 1.0, Auto := 1, DeltaT := 1.0);   // mcv temp pid
   Temp_PID1 : PID_ENHANCED := (PVEUMax := 100.0, SPHLimit := 100.0, RatioProg := 1.0, RatioOper := 1.0, RatioHLimit := 1.0, RatioLLimit := 1.0, CVEUMax := 100.0, CVHLimit := 100.0, PVEDerivative := 1, RTSTime := 1);   // mcv temp pid
   Temp_PID2 : PID_ENHANCED := (PVEUMax := 100.0, SPHLimit := 100.0, RatioProg := 1.0, RatioOper := 1.0, RatioHLimit := 1.0, RatioLLimit := 1.0, CVEUMax := 100.0, CVHLimit := 100.0, PVEDerivative := 1, RTSTime := 1);   // mcv temp pid
   Temp_Scaler : SCALE := (InRawMax := 100.0, InEUMax := 15.0);
   TempEUMax : REAL := 15.0;
   TempEUMin : REAL;
   TempOffOns : BOOL := 1;
   TempOnOns : BOOL;
   TempRawMax : REAL := 100.0;
   TempRawMin : REAL;
   Test_Temp_Raw : REAL := 95.0;
   TOT101 : TOTALIZER := (TimeBase := 1, Gain := 1.0, ProgStopReq := 1, RTSTime := 1, Total := 82085.13, OldTotal := 9317.5, ProgOper := 1, TargetFlag := 1, TargetDev1Flag := 1, TargetDev2Flag := 1, LowInCutoffFlag := 1, DeltaT := 0.1);
   TOT102 : TOTALIZER := (TimeBase := 1, Gain := 1.0, ProgStopReq := 1, RTSTime := 1, Total := 43741.168, ProgOper := 1, TargetFlag := 1, TargetDev1Flag := 1, TargetDev2Flag := 1, LowInCutoffFlag := 1, DeltaT := 0.1);
   TOT1021 : TOTALIZER := (Gain := 1.0, RTSTime := 1);
   TOT1022 : TOTALIZER := (Gain := 1.0, RTSTime := 1);
   TOT1023 : TOTALIZER := (Gain := 1.0, RTSTime := 1);
   TOT103 : TOTALIZER := (TimeBase := 1, Gain := 1.0, ProgStopReq := 1, RTSTime := 1, Total := 3248.3599, OldTotal := 5510706.5, ProgOper := 1, TargetFlag := 1, TargetDev1Flag := 1, TargetDev2Flag := 1, LowInCutoffFlag := 1, DeltaT := 0.1);
   TOT104 : TOTALIZER := (TimeBase := 1, Gain := 1.0, ProgStopReq := 1, RTSTime := 1, Total := 4920184.0, ProgOper := 1, TargetFlag := 1, TargetDev1Flag := 1, TargetDev2Flag := 1, LowInCutoffFlag := 1, DeltaT := 0.1);
   TOT105 : TOTALIZER := (TimeBase := 1, Gain := 1.0, ProgStopReq := 1, RTSTime := 1, Total := 288757.94, ProgOper := 1, TargetFlag := 1, TargetDev1Flag := 1, TargetDev2Flag := 1, LowInCutoffFlag := 1, DeltaT := 0.1);
   Total_Gas_Flow_Limit : REAL := 3.0;
   TotalFlowSP : REAL := 6.0;
   TT700 : P_AInAdv := (Inp_PV := 95.0, Inp_HiHiGate := 1, Inp_HiGate := 1, Inp_LoGate := 1, Inp_LoLoGate := 1, Inp_HiRoCGate := 1, Inp_HiDevGate := 1, Inp_LoDevGate := 1, Inp_FailGate := 1, Cfg_PVDecPlcs := 2, Cfg_HasHiHiAlm := 1, Cfg_HasHiAlm := 1, Cfg_HasLoAlm := 1, Cfg_HasLoLoAlm := 1, Cfg_HiHiAckReqd := 1, Cfg_HiAckReqd := 1, Cfg_LoAckReqd := 1, Cfg_LoLoAckReqd := 1, Cfg_HiRoCAckReqd := 1, Cfg_HiDevAckReqd := 1, Cfg_LoDevAckReqd := 1, Cfg_FailAckReqd := 1, Cfg_HiHiSeverity := 1000, Cfg_HiSeverity := 500, Cfg_LoSeverity := 500, Cfg_LoLoSeverity := 750, Cfg_HiRoCSeverity := 500, Cfg_HiDevSeverity := 500, Cfg_LoDevSeverity := 500, Cfg_FailSeverity := 1000, Cfg_InpRawMax := 100.0, Cfg_PVEUMax := 100.0, Cfg_RateTime := 1.0, Cfg_CtrlHiHiLim := 1.5e+38, Cfg_CtrlHiHiDB := 1.0, Cfg_CtrlHiLim := 1.5e+38, Cfg_CtrlHiDB := 1.0, Cfg_CtrlLoLim := -1.5e+38, Cfg_CtrlLoDB := 1.0, Cfg_CtrlLoLoLim := -1.5e+38, Cfg_CtrlLoLoDB := 1.0, Cfg_HiHiLim := 100.0, Cfg_HiLim := 1.5e+38, Cfg_HiDB := 1.0, Cfg_LoLim := -1.5e+38, Cfg_LoDB := 1.0, Cfg_LoLoLim := -1.5e+38, Cfg_LoLoDB := 1.0, Cfg_HiRoCLim := 1.5e+38, Cfg_HiRoCDB := 1.0, Cfg_HiDevLim := 1.5e+38, Cfg_HiDevDB := 1.0, Cfg_LoDevLim := -1.5e+38, Cfg_LoDevDB := 1.0, Cfg_FailHiLim := 103.958336, Cfg_FailLoLim := -2.0833333, Cfg_FailDB := 0.41666666, MSet_SubstPV := 95.0, Set_SimPV := 95.0, Val := 95.0,
        Val_InpPV := 95.0, Val_PVMinCapt := 95.0, Val_PVMaxCapt := 95.0, Val_PVEUMax := 100.0, SrcQ_IO := 1, SrcQ := 1, Val_NotifyAll := 1, Val_UnackAlmC := 1, Sts_RdyAck := 1, Sts_HiHiGate := 1, Sts_HiGate := 1, Ack_Hi := 1, Sts_LoGate := 1, Ack_Lo := 1, Sts_LoLoGate := 1, Ack_LoLo := 1, Sts_HiRoCGate := 1, Ack_HiRoC := 1, Sts_HiDevGate := 1, Ack_HiDev := 1, Sts_LoDevGate := 1, Ack_LoDev := 1, Sts_FailGate := 1, Ack_Fail := 1);   // Temperature Transmitter
   TT700_1Point_Complete : BOOL;
   TT700_1Point_Offset : REAL := -73.0;
   TT700_1Point_Running : BOOL;
   TT700_2Point_Complete : BOOL;
   TT700_2PointAccept : BOOL;
   TT700_Accept1Point : BOOL;
   TT700_CalClear : BOOL;
   TT700_MaxCfg : REAL := 100.0;
   TT700_MinCfg : REAL;
   TT700_NewMax : REAL := 102.0;
   TT700_NewMin : REAL := 2.0;
   TT700_RawMax : REAL := 95.0;
   TT700_RawMin : REAL := 5.0;
   TT700_RawRange : REAL := 90.0;
   TT700_Ref1Point : REAL := 22.0;
   TT700_RefMax : REAL := 85.0;
   TT700_RefMin : REAL := 10.0;
   TT700_RefRange : REAL := 75.0;
   WT701 : P_AInAdv := (Inp_HiHiGate := 1, Inp_HiGate := 1, Inp_LoGate := 1, Inp_LoLoGate := 1, Inp_HiRoCGate := 1, Inp_HiDevGate := 1, Inp_LoDevGate := 1, Inp_FailGate := 1, Cfg_PVDecPlcs := 2, Cfg_HasHiHiAlm := 1, Cfg_HasHiAlm := 1, Cfg_HasLoAlm := 1, Cfg_HasLoLoAlm := 1, Cfg_HiHiAckReqd := 1, Cfg_HiAckReqd := 1, Cfg_LoAckReqd := 1, Cfg_LoLoAckReqd := 1, Cfg_HiRoCAckReqd := 1, Cfg_HiDevAckReqd := 1, Cfg_LoDevAckReqd := 1, Cfg_FailAckReqd := 1, Cfg_HiHiSeverity := 750, Cfg_HiSeverity := 500, Cfg_LoSeverity := 500, Cfg_LoLoSeverity := 750, Cfg_HiRoCSeverity := 500, Cfg_HiDevSeverity := 500, Cfg_LoDevSeverity := 500, Cfg_FailSeverity := 1000, Cfg_InpRawMax := 100.0, Cfg_PVEUMax := 60.0, Cfg_RateTime := 1.0, Cfg_CtrlHiHiLim := 1.5e+38, Cfg_CtrlHiHiDB := 1.0, Cfg_CtrlHiLim := 1.5e+38, Cfg_CtrlHiDB := 1.0, Cfg_CtrlLoLim := -1.5e+38, Cfg_CtrlLoDB := 1.0, Cfg_CtrlLoLoLim := -1.5e+38, Cfg_CtrlLoLoDB := 1.0, Cfg_HiHiLim := 20.0, Cfg_HiHiDB := 1.0, Cfg_HiLim := 18.0, Cfg_HiDB := 1.0, Cfg_LoLim := 1.0, Cfg_LoDB := 1.0, Cfg_LoLoDB := 1.0, Cfg_HiRoCLim := 1.5e+38, Cfg_HiRoCDB := 1.0, Cfg_HiDevLim := 1.5e+38, Cfg_HiDevDB := 1.0, Cfg_LoDevLim := -1.5e+38, Cfg_LoDevDB := 1.0, Cfg_FailHiLim := 103.958336, Cfg_FailLoLim := -2.0833333, Cfg_FailDB := 0.41666666, MSet_SubstPV := 5.0, Val := 5.0, Val_PVMinCapt := 5.0, Val_PVMaxCapt := 5.0,
        Val_PVEUMax := 60.0, SrcQ_IO := 1, SrcQ := 18, Val_NotifyAll := 1, Val_UnackAlmC := 1, Sts_SubstPV := 1, Sts_MaintByp := 1, Sts_RdyAck := 1, Sts_HiHiGate := 1, Ack_HiHi := 1, Sts_HiGate := 1, Ack_Hi := 1, Sts_LoGate := 1, Ack_Lo := 1, Sts_LoLoGate := 1, Sts_HiRoCGate := 1, Ack_HiRoC := 1, Sts_HiDevGate := 1, Ack_HiDev := 1, Sts_LoDevGate := 1, Ack_LoDev := 1, Sts_FailGate := 1, Ack_Fail := 1);   // Media Scale
   WT702 : P_AInAdv := (Inp_HiHiGate := 1, Inp_HiGate := 1, Inp_LoGate := 1, Inp_LoLoGate := 1, Inp_HiRoCGate := 1, Inp_HiDevGate := 1, Inp_LoDevGate := 1, Inp_FailGate := 1, Cfg_PVDecPlcs := 2, Cfg_HasHiHiAlm := 1, Cfg_HasHiAlm := 1, Cfg_HasLoAlm := 1, Cfg_HasLoLoAlm := 1, Cfg_HiHiAckReqd := 1, Cfg_HiAckReqd := 1, Cfg_LoAckReqd := 1, Cfg_LoLoAckReqd := 1, Cfg_HiRoCAckReqd := 1, Cfg_HiDevAckReqd := 1, Cfg_LoDevAckReqd := 1, Cfg_FailAckReqd := 1, Cfg_HiHiSeverity := 750, Cfg_HiSeverity := 500, Cfg_LoSeverity := 500, Cfg_LoLoSeverity := 750, Cfg_HiRoCSeverity := 500, Cfg_HiDevSeverity := 500, Cfg_LoDevSeverity := 500, Cfg_FailSeverity := 1000, Cfg_InpRawMax := 100.0, Cfg_PVEUMax := 100.0, Cfg_RateTime := 1.0, Cfg_CtrlHiHiLim := 1.5e+38, Cfg_CtrlHiHiDB := 1.0, Cfg_CtrlHiLim := 1.5e+38, Cfg_CtrlHiDB := 1.0, Cfg_CtrlLoLim := -1.5e+38, Cfg_CtrlLoDB := 1.0, Cfg_CtrlLoLoLim := -1.5e+38, Cfg_CtrlLoLoDB := 1.0, Cfg_HiHiLim := 25.0, Cfg_HiLim := 13.0, Cfg_LoLim := 2.0, Cfg_LoLoLim := 1.0, Cfg_HiRoCLim := 1.5e+38, Cfg_HiRoCDB := 1.0, Cfg_HiDevLim := 1.5e+38, Cfg_HiDevDB := 1.0, Cfg_LoDevLim := -1.5e+38, Cfg_LoDevDB := 1.0, Cfg_FailHiLim := 103.958336, Cfg_FailLoLim := -2.0833333, Cfg_FailDB := 0.41666666, MSet_SubstPV := 3.0, Val := 3.0, Val_PVMinCapt := 3.0, Val_PVMaxCapt := 3.0, Val_PVEUMax := 100.0, SrcQ_IO := 1, SrcQ := 18,
        Val_NotifyAll := 1, Val_UnackAlmC := 4, Sts_SubstPV := 1, Sts_MaintByp := 1, Sts_RdyAck := 1, Sts_HiHiGate := 1, Sts_HiGate := 1, Sts_LoGate := 1, Sts_LoLoGate := 1, Sts_HiRoCGate := 1, Ack_HiRoC := 1, Sts_HiDevGate := 1, Ack_HiDev := 1, Sts_LoDevGate := 1, Ack_LoDev := 1, Sts_FailGate := 1, Ack_Fail := 1);   // MCV Weight
   WT703 : P_AInAdv := (Inp_HiHiGate := 1, Inp_HiGate := 1, Inp_LoGate := 1, Inp_LoLoGate := 1, Inp_HiRoCGate := 1, Inp_HiDevGate := 1, Inp_LoDevGate := 1, Inp_FailGate := 1, Cfg_PVDecPlcs := 2, Cfg_HasHiHiAlm := 1, Cfg_HasHiAlm := 1, Cfg_HasLoAlm := 1, Cfg_HasLoLoAlm := 1, Cfg_HiHiAckReqd := 1, Cfg_HiAckReqd := 1, Cfg_LoAckReqd := 1, Cfg_LoLoAckReqd := 1, Cfg_HiRoCAckReqd := 1, Cfg_HiDevAckReqd := 1, Cfg_LoDevAckReqd := 1, Cfg_FailAckReqd := 1, Cfg_HiHiSeverity := 750, Cfg_HiSeverity := 500, Cfg_LoSeverity := 500, Cfg_LoLoSeverity := 750, Cfg_HiRoCSeverity := 500, Cfg_HiDevSeverity := 500, Cfg_LoDevSeverity := 500, Cfg_FailSeverity := 1000, Cfg_InpRawMax := 100.0, Cfg_PVEUMax := 60.0, Cfg_RateTime := 1.0, Cfg_CtrlHiHiLim := 1.5e+38, Cfg_CtrlHiHiDB := 1.0, Cfg_CtrlHiLim := 1.5e+38, Cfg_CtrlHiDB := 1.0, Cfg_CtrlLoLim := -1.5e+38, Cfg_CtrlLoDB := 1.0, Cfg_CtrlLoLoLim := -1.5e+38, Cfg_CtrlLoLoDB := 1.0, Cfg_HiHiLim := 20.0, Cfg_HiHiDB := 1.0, Cfg_HiLim := 18.0, Cfg_HiDB := 1.0, Cfg_LoLim := 1.0, Cfg_LoDB := 1.0, Cfg_LoLoLim := 1.0, Cfg_HiRoCLim := 1.5e+38, Cfg_HiRoCDB := 1.0, Cfg_HiDevLim := 1.5e+38, Cfg_HiDevDB := 1.0, Cfg_LoDevLim := -1.5e+38, Cfg_LoDevDB := 1.0, Cfg_FailHiLim := 103.958336, Cfg_FailLoLim := -2.0833333, Cfg_FailDB := 0.41666666, MSet_SubstPV := 2.0, Val := 2.0, Val_PVMinCapt := 2.0, Val_PVMaxCapt := 2.0,
        Val_PVEUMax := 60.0, SrcQ_IO := 1, SrcQ := 18, Val_NotifyAll := 1, Val_UnackAlmC := 2, Sts_SubstPV := 1, Sts_MaintByp := 1, Sts_RdyAck := 1, Sts_HiHiGate := 1, Sts_HiGate := 1, Sts_LoGate := 1, Ack_Lo := 1, Sts_LoLoGate := 1, Ack_LoLo := 1, Sts_HiRoCGate := 1, Ack_HiRoC := 1, Sts_HiDevGate := 1, Ack_HiDev := 1, Sts_LoDevGate := 1, Ack_LoDev := 1, Sts_FailGate := 1, Ack_Fail := 1);   // Spent Media/Harvest Scale
END_VAR
